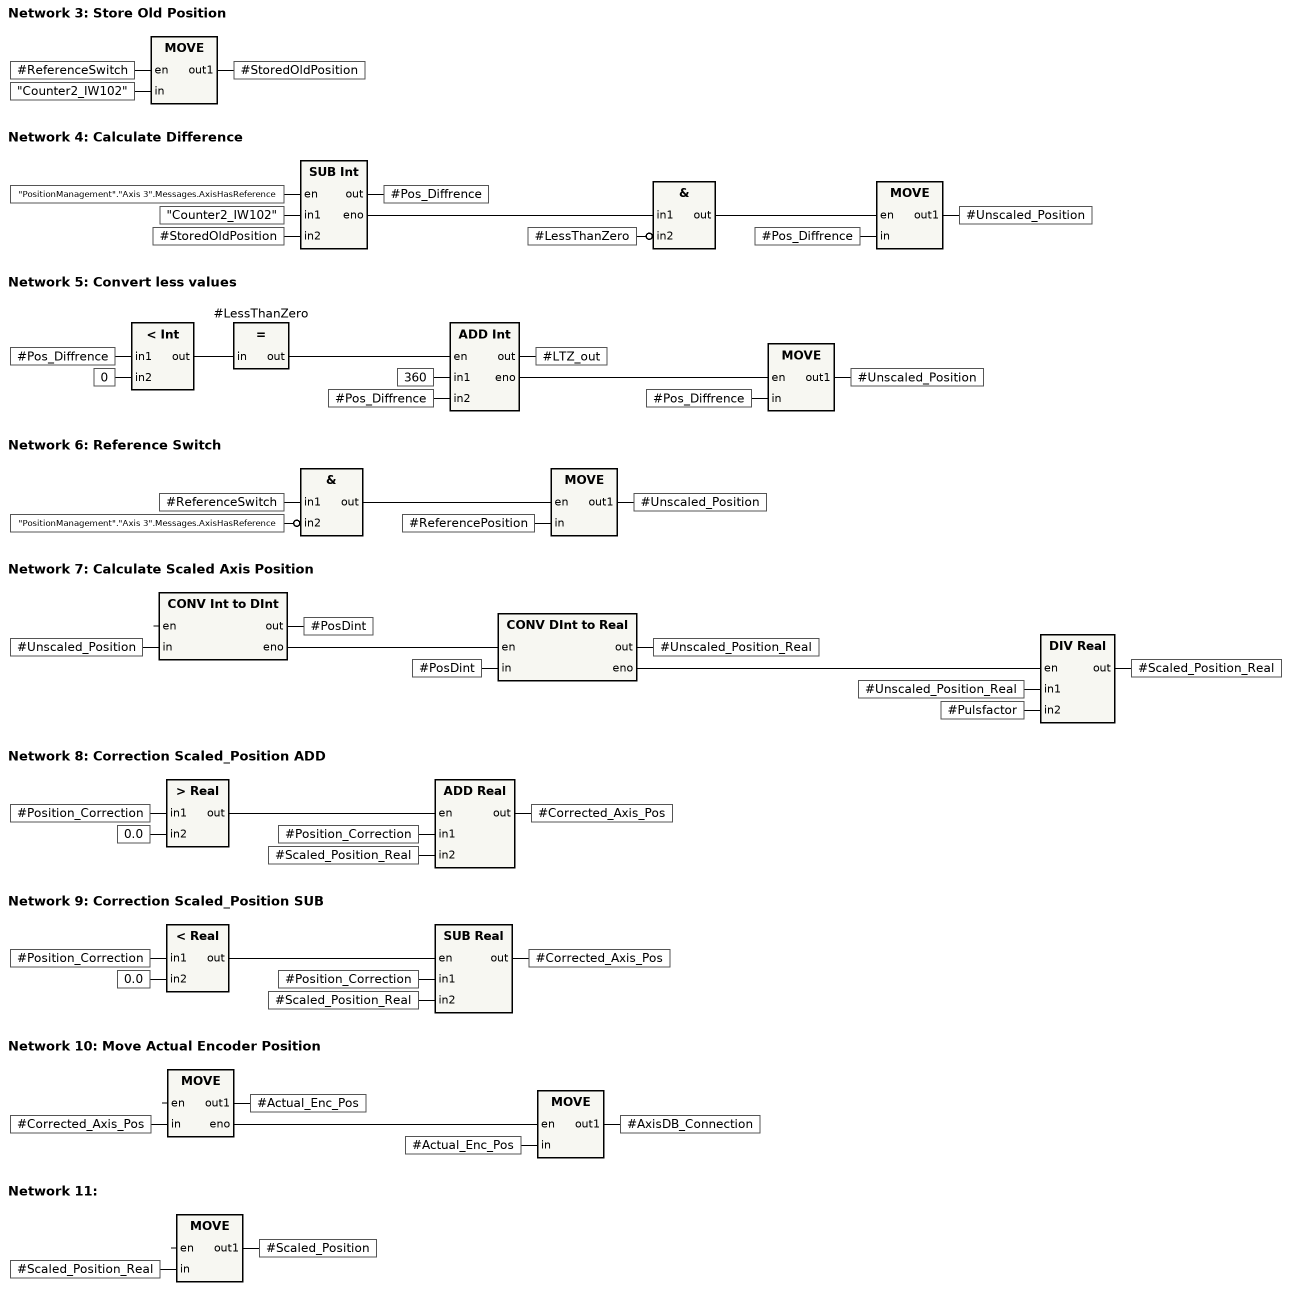
   IF #ReferenceSwitch THEN #StoredOldPosition := "Counter2_IW102"; END_IF;
END_REGION

REGION Network 4: Calculate Difference
   // ENO of a box is taken as its EN; it also drops when the box reports an error
   IF "PositionManagement"."Axis 3".Messages.AxisHasReference THEN
       #Pos_Diffrence := "Counter2_IW102" - #StoredOldPosition;
   END_IF;
   IF "PositionManagement"."Axis 3".Messages.AxisHasReference AND NOT #LessThanZero THEN
       #Unscaled_Position := #Pos_Diffrence;
   END_IF;
END_REGION

REGION Network 5: Convert less values
   // ENO of a box is taken as its EN; it also drops when the box reports an error
   #LessThanZero := #Pos_Diffrence < 0;
   IF #LessThanZero THEN
       #LTZ_out := 360 + #Pos_Diffrence;
       #Unscaled_Position := #Pos_Diffrence;
   END_IF;
END_REGION

REGION Network 6: Reference Switch
   IF #ReferenceSwitch AND NOT "PositionManagement"."Axis 3".Messages.AxisHasReference THEN
       #Unscaled_Position := #ReferencePosition;
   END_IF;
END_REGION

REGION Network 7: Calculate Scaled Axis Position
   // ENO of a box is taken as its EN; it also drops when the box reports an error
   #PosDint := INT_TO_DINT(#Unscaled_Position);
   #Unscaled_Position_Real := DINT_TO_REAL(#PosDint);
   #Scaled_Position_Real := #Unscaled_Position_Real / #Pulsfactor;
END_REGION

REGION Network 8: Correction Scaled_Position ADD
   IF #Position_Correction > 0.0 THEN
       #Corrected_Axis_Pos := #Position_Correction + #Scaled_Position_Real;
   END_IF;
END_REGION

REGION Network 9: Correction Scaled_Position SUB
   IF #Position_Correction < 0.0 THEN
       #Corrected_Axis_Pos := #Position_Correction - #Scaled_Position_Real;
   END_IF;
END_REGION

REGION Network 10: Move Actual Encoder Position
   // ENO of a box is taken as its EN; it also drops when the box reports an error
   #Actual_Enc_Pos := #Corrected_Axis_Pos;
   #AxisDB_Connection := #Actual_Enc_Pos;
END_REGION

REGION Network 11
   #Scaled_Position := #Scaled_Position_Real;
END_REGION
END_FUNCTION

FUNCTION_BLOCK "MC_Move"   // FB10, FBD
TITLE = MC_Move
VERSION : 0.1
// Block moves an Axis to an Desired Position, this block comes with the brake feature. When the axis is on position it keeps the brake for a time. You can set the time in the Brake Time field.
// stored: AutoNumber true, IsIECCheckEnabled false, UDAEnableTagReadback false
   VAR_INPUT
      Start : Bool;
      "Desired Position" : Real;
      "Speed (50-75%)" : Int;
      "Brake on Position" : Bool;
      Acceleration : Real;
      Deacceleration : Real;
      "Drive Ready" : Bool;
      "Drive On Position" : Bool;
      "Brake Time" : Time := T#500ms;
      "Safety OK" : Bool;
   END_VAR
   VAR_OUTPUT
      Go : Bool;
      "Desired Position Out" : Real;
      "Speed Output" : Int;
      "Acceleration Out" : Real;
      "Deacceleration Out" : Real;
      "Brake Out" : Bool;
   END_VAR
   VAR_TEMP
      SR_1 : Bool;
   END_VAR
BEGIN

REGION Network 1: Start - Go To Position + Speed
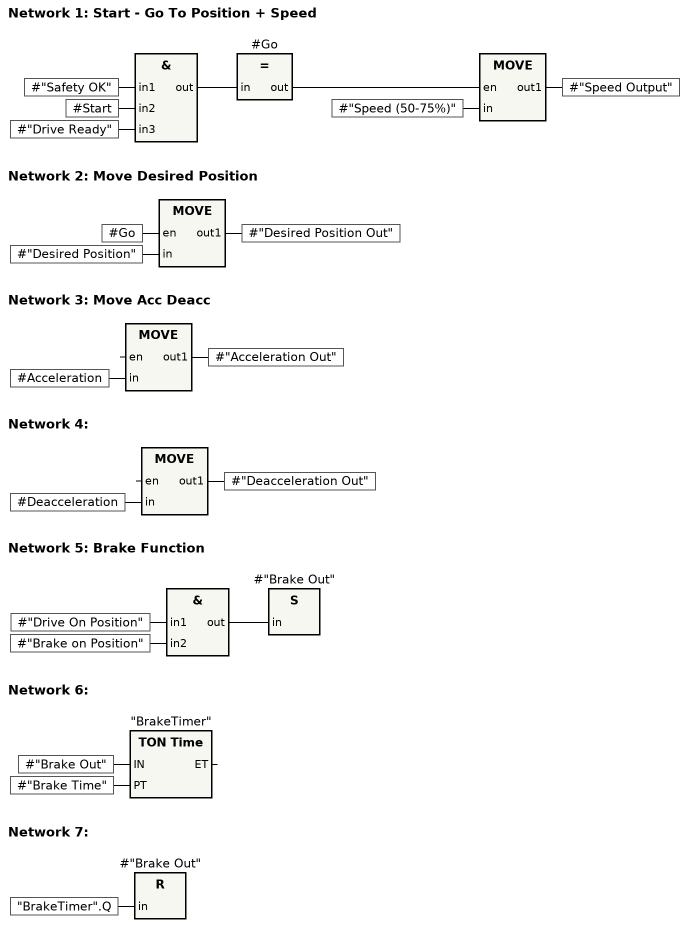
   #Go := #"Safety OK" AND #Start AND #"Drive Ready";
   IF #Go THEN #"Speed Output" := #"Speed (50-75%)"; END_IF;
END_REGION

REGION Network 2: Move Desired Position
   IF #Go THEN #"Desired Position Out" := #"Desired Position"; END_IF;
END_REGION

REGION Network 3: Move Acc Deacc
   #"Acceleration Out" := #Acceleration;
END_REGION

REGION Network 4
   #"Deacceleration Out" := #Deacceleration;
END_REGION

REGION Network 5: Brake Function
   IF #"Drive On Position" AND #"Brake on Position" THEN #"Brake Out" := TRUE; END_IF;
END_REGION

REGION Network 6
   "BrakeTimer".TON(IN := #"Brake Out", PT := #"Brake Time");
END_REGION

REGION Network 7
   IF "BrakeTimer".Q THEN #"Brake Out" := FALSE; END_IF;
END_REGION
END_FUNCTION_BLOCK

FUNCTION_BLOCK "MC_Jog"   // FB11, FBD
TITLE = MC_Jog
VERSION : 0.1
// With this block you can Jog an Axis manual, you can set the speed on 25%, 50% or 75%. It also has an brake functionality, when you set Brake to true, it holds the brake for 2 seconds, then releases it.
// stored: AutoNumber true, IsIECCheckEnabled false, UDAEnableTagReadback false
   VAR_INPUT
      "Jog Forward" : Bool;
      "Jog Backward" : Bool;
      Speed : Int;
      Brake : Bool;
   END_VAR
   VAR_OUTPUT
      "Drive Fwd Output" : Bool;
      "Drive Rev Output" : Bool;
      "Drive Speed Output" : Int;
      "Drive Brake Output" : Bool;
   END_VAR
BEGIN

REGION Network 1: Manual Control
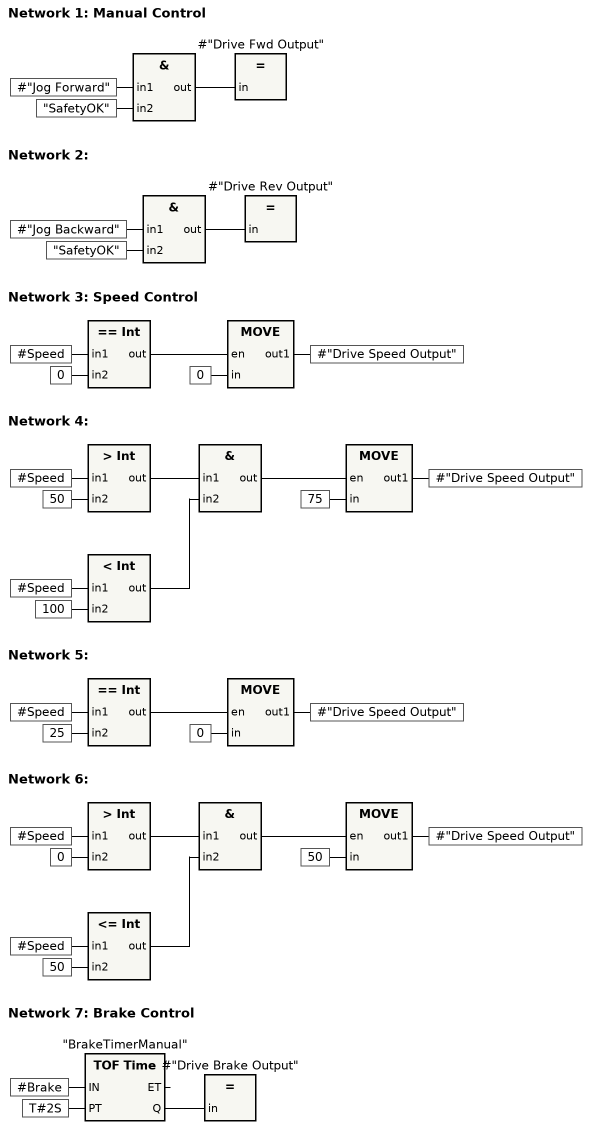
   #"Drive Fwd Output" := #"Jog Forward" AND "SafetyOK";
END_REGION

REGION Network 2
   #"Drive Rev Output" := #"Jog Backward" AND "SafetyOK";
END_REGION

REGION Network 3: Speed Control
   IF #Speed = 0 THEN #"Drive Speed Output" := 0; END_IF;
END_REGION

REGION Network 4
   IF (#Speed > 50) AND (#Speed < 100) THEN #"Drive Speed Output" := 75; END_IF;
END_REGION

REGION Network 5
   IF #Speed = 25 THEN #"Drive Speed Output" := 0; END_IF;
END_REGION

REGION Network 6
   IF (#Speed > 0) AND (#Speed <= 50) THEN #"Drive Speed Output" := 50; END_IF;
END_REGION

REGION Network 7: Brake Control
   "BrakeTimerManual".TOF(IN := #Brake, PT := T#2S);
   #"Drive Brake Output" := "BrakeTimerManual".Q;
END_REGION
END_FUNCTION_BLOCK

FUNCTION_BLOCK "ProductBuffer"
{ S7_Optimized_Access := 'FALSE' }
VERSION : 0.1
   VAR_INPUT 
      SensorInput : Bool;
      TimeDelay : Time;
      TriggerFeedback : Bool;
   END_VAR

   VAR_OUTPUT 
      TriggerMovement : Bool;
      ProductCount : Int;
   END_VAR

   VAR 
      PrevSensor : Bool;
      DelayTimer {InstructionName := 'TON'; LibVersion := '1.0'; S7_SetPoint := 'False'} : TON;
      MovementActive { S7_SetPoint := 'True'} : Bool;
   END_VAR


BEGIN
	// Flankdetectie op sensor
	IF #SensorInput AND NOT #PrevSensor THEN
	    IF #ProductCount < 32767 THEN
	        #ProductCount := #ProductCount + 1;
	    END_IF;
	END_IF;
	#PrevSensor := #SensorInput;
	
	// Timer mag alleen lopen als:
	// - Er producten zijn
	// - Er geen beweging actief is
	IF (#ProductCount > 0) AND (NOT #MovementActive) THEN
	    #DelayTimer(IN := TRUE,
	                PT := #TimeDelay);
	ELSE
	    #DelayTimer(IN := FALSE,
	                PT := #TimeDelay);
	END_IF;
	
	// Als de timer klaar is → activeer beweging en zet MovementActive
	IF #DelayTimer.Q THEN
	    #TriggerMovement := TRUE;
	    #MovementActive := TRUE;
	    #ProductCount := #ProductCount - 1;
	    #DelayTimer(IN := FALSE,
	                PT := #TimeDelay); // Reset timer
	END_IF;
	
	// Wacht op TriggerFeedback om TriggerMovement terug laag te zetten
	IF #MovementActive AND #TriggerFeedback THEN
	    #TriggerMovement := FALSE;
	    #MovementActive := FALSE;
	END_IF;
	
END_FUNCTION_BLOCK

FUNCTION_BLOCK "ProductBuffer_V3"
{ S7_Optimized_Access := 'FALSE' }
VERSION : 0.1
   VAR_INPUT 
      SensorInput : Bool;   // Sensor aan begin band
      EncoderPosition : DInt;   // Koppel aan Encoder Data Instance
      TriggerDistance : DInt;   // Gewenste Afstand Product voor trigger
      TriggerFeedback : Bool;
   END_VAR

   VAR_OUTPUT 
      TriggerMovement : Bool;   // Trigger Start Movement
      ProductCount : Int;   // Count products in buffer
   END_VAR

   VAR 
      ProductBuffer { S7_SetPoint := 'False'} : Array[0..9] of "ProductTrack";
      PrevSensor { S7_SetPoint := 'True'} : Bool;
      MovementActive : Bool;
      i : Int;
      Distance : DInt;
   END_VAR


BEGIN
	// 1️⃣ Flankdetectie - detecteer nieuw product
	IF #SensorInput AND NOT #PrevSensor THEN
	    FOR #i := 0 TO 9 DO
	        IF NOT #ProductBuffer[#i].Active THEN
	            #ProductBuffer[#i].StartPosition := #EncoderPosition;
	            #ProductBuffer[#i].Active := TRUE;
	            EXIT;
	        END_IF;
	    END_FOR;
	END_IF;
	#PrevSensor := #SensorInput;
	
	// 2️⃣ Tel actieve producten
	#ProductCount := 0;
	FOR #i := 0 TO 9 DO
	    IF #ProductBuffer[#i].Active THEN
	        #ProductCount := #ProductCount + 1;
	    END_IF;
	END_FOR;
	
	// 3️⃣ Zoek eerste product dat zijn afstand heeft afgelegd
	IF NOT #MovementActive THEN
	    FOR #i := 0 TO 9 DO
	        IF #ProductBuffer[#i].Active THEN
	            #Distance := #ProductBuffer[#i].StartPosition - #EncoderPosition;
	            IF #Distance >= #TriggerDistance THEN
	                #TriggerMovement := TRUE;
	                #MovementActive := TRUE;
	                #ProductBuffer[#i].Active := FALSE;
	                EXIT;
	            END_IF;
	        END_IF;
	    END_FOR;
	END_IF;
	
	// 4️⃣ Wacht op feedback om beweging af te ronden
	IF #MovementActive AND #TriggerFeedback THEN
	    #TriggerMovement := FALSE;
	    #MovementActive := FALSE;
	END_IF;
	
END_FUNCTION_BLOCK

FUNCTION_BLOCK "FB_EncoderFeedback_Lineair"   // FB21, FBD
TITLE = Encoder Feedback Function Block Lineair Axis
VERSION : 0.1
// stored: AutoNumber true, IsIECCheckEnabled false, UDAEnableTagReadback false
   VAR_INPUT
      CounterTag { ExternalVisible := 'False'; ExternalWritable := 'False'} : DInt;   // Connect to the CounterTag IW102
      Position_Offset { ExternalVisible := 'False'; ExternalWritable := 'False'} : Real;   // Fill in the tolerance, when the axis approves the position. Above or below the desired position
      Pulsfactor { ExternalVisible := 'False'; ExternalWritable := 'False'} : Real;   // Number of pulses after an defined distance of the axis.
      Position_Correction { ExternalVisible := 'False'; ExternalWritable := 'False'} : Real;   // Small Position Correction for the Axis
      ReferenceRun_Command { ExternalVisible := 'False'; ExternalWritable := 'False'} : Bool;   // Command of starting the referencerun
      ReferenceSwitch { ExternalVisible := 'False'; ExternalWritable := 'False'} : Bool;   // ReferenceSwitch Mounted on Axis
      ReferencePosition { ExternalVisible := 'False'; ExternalWritable := 'False'} : Int;   // Position where the index puls of the reference switch enters.
      WrappingPosition : Real;   // Max Position of the axis. From there the position
   END_VAR
   VAR_OUTPUT
      Scaled_Position { ExternalVisible := 'False'; ExternalWritable := 'False'} : Real;   // Scaled Position scaled with Pulsfactor
      Actual_Enc_Pos { ExternalVisible := 'False'; ExternalWritable := 'False'} : Real;   // Actual Encoder Position
      AxisDB_Connection { ExternalVisible := 'False'; ExternalWritable := 'False'} : Real;   // Connection with Axis DB connection
   END_VAR
   VAR_TEMP
      Corrected_Axis_Pos : Real;
      Unscaled_Position : DInt;   // Unscaled Position of the Encoder
      Unsc2 : DInt;   // Unsc 2 position
      Act_Enc_Pos_Int : DInt;
      Scaled_Position_Real : Real;
      PosDint : DInt;
      Unscaled_Position_Real : Real;
      InternalCounter : DInt;
      CalDifCounter : DInt;
      Pos_Storage : DInt;
      Pos_Diffrence : DInt;
      Add_Pos : DInt;
      Sub_Pos : DInt;
      LessThanZero : Bool;
      LTZ_out : DInt;
      WrappedPosTemp : Real;
      DivWrapping : Real;
      TruncWrapping : DInt;
      TruncWrappingReal : Real;
      ScaledBackWrapping : Real;
      AxisPosTooHigh : Bool;
      WeDontUseThisAnymore : Bool;
      SRMOve : Bool;
      noreset : Bool;
      nououtput : Bool;
      OverflowProtectPulses : DInt;
      SegmentCounter : DInt;
   END_VAR
BEGIN

REGION Network 1: Overflow Buffer FB
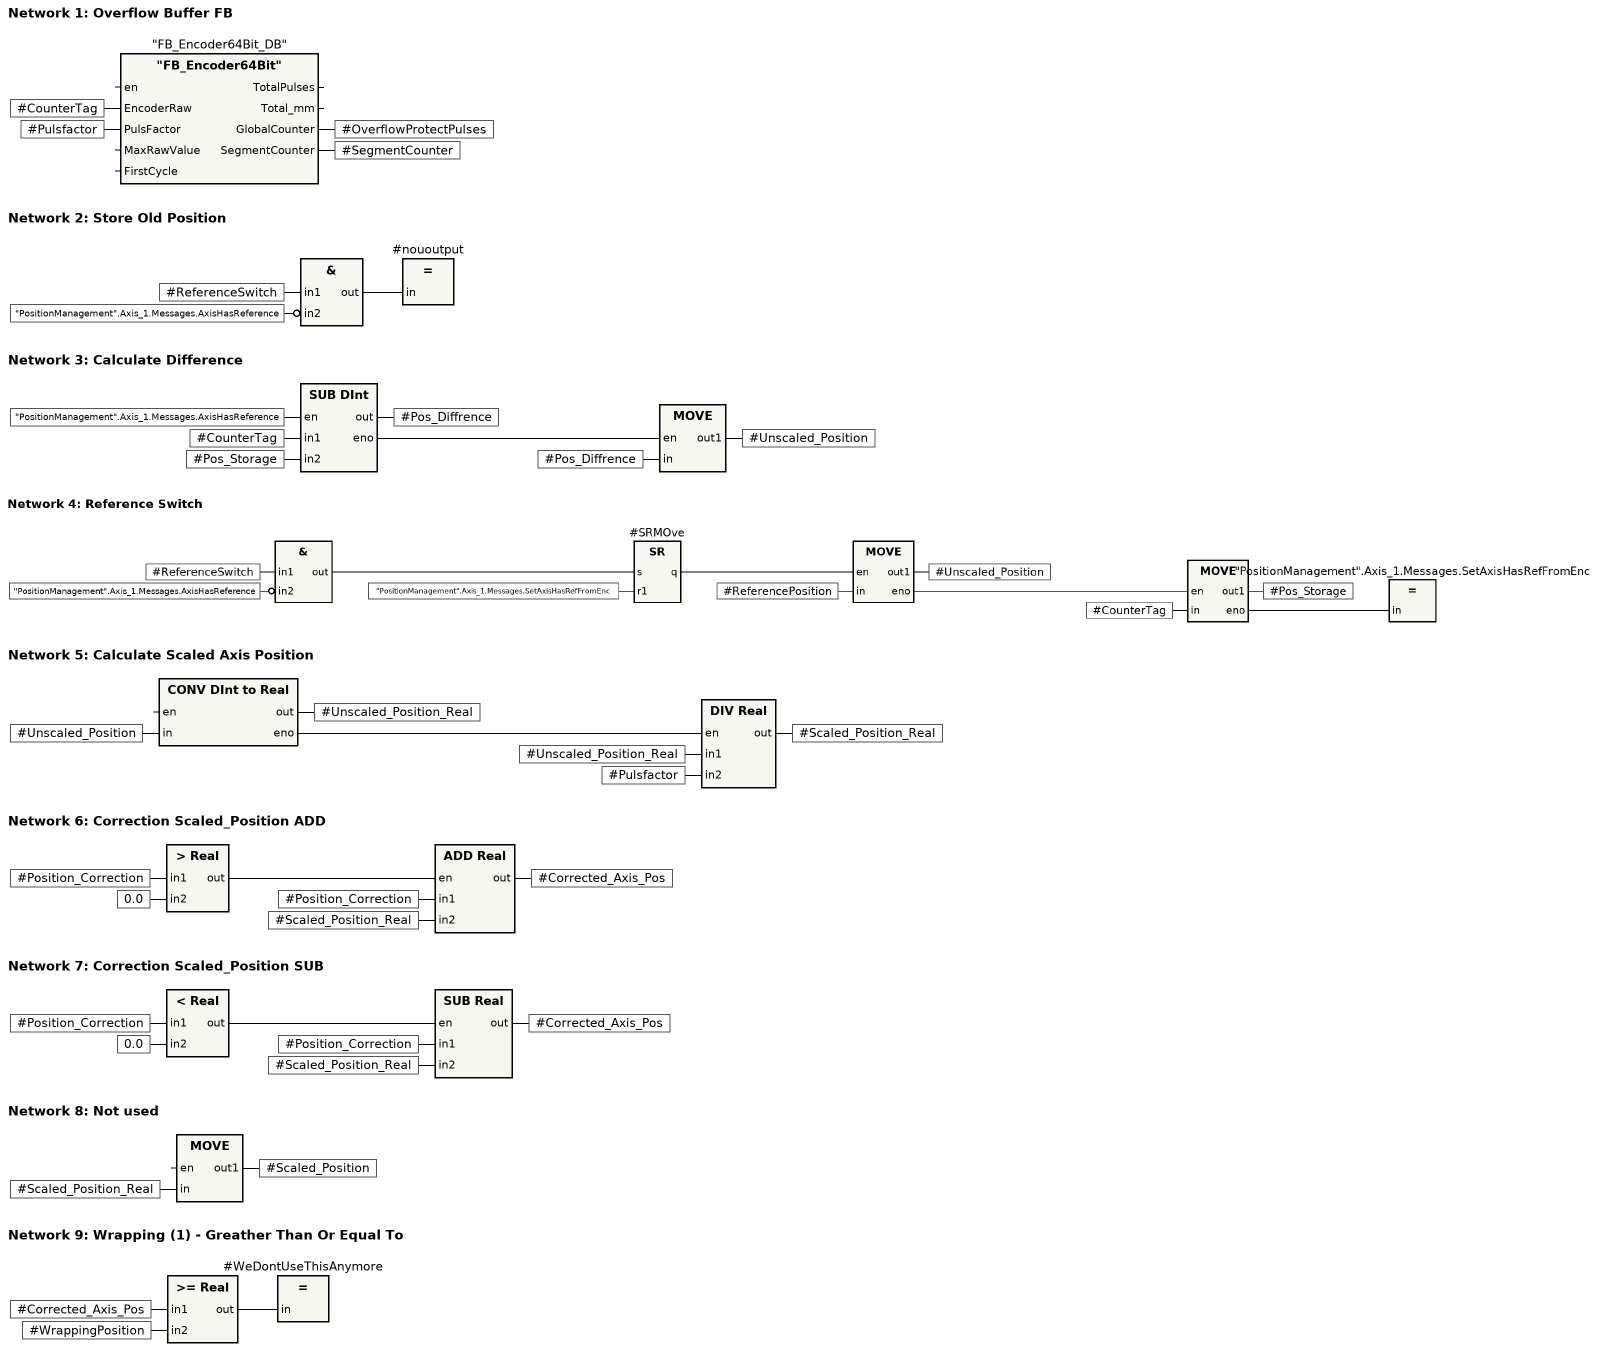
   "FB_Encoder64Bit_DB"(EncoderRaw := #CounterTag,   // "FB_Encoder64Bit"
                        PulsFactor := #Pulsfactor,
                        GlobalCounter => #OverflowProtectPulses,
                        SegmentCounter => #SegmentCounter);
END_REGION

REGION Network 2: Store Old Position
   #nououtput := #ReferenceSwitch AND NOT "PositionManagement".Axis_1.Messages.AxisHasReference;
END_REGION

REGION Network 3: Calculate Difference
   // ENO of a box is taken as its EN; it also drops when the box reports an error
   IF "PositionManagement".Axis_1.Messages.AxisHasReference THEN
       #Pos_Diffrence := #CounterTag - #Pos_Storage;
       #Unscaled_Position := #Pos_Diffrence;
   END_IF;
END_REGION

REGION Network 4: Reference Switch
   // ENO of a box is taken as its EN; it also drops when the box reports an error
   IF #ReferenceSwitch AND NOT "PositionManagement".Axis_1.Messages.AxisHasReference THEN
       #SRMOve := TRUE;   // SR flip-flop
   END_IF;
   IF "PositionManagement".Axis_1.Messages.SetAxisHasRefFromEnc THEN #SRMOve := FALSE; END_IF;
   IF #SRMOve THEN
       #Unscaled_Position := #ReferencePosition;
       #Pos_Storage := #CounterTag;
   END_IF;
   "PositionManagement".Axis_1.Messages.SetAxisHasRefFromEnc := #SRMOve;
END_REGION

REGION Network 5: Calculate Scaled Axis Position
   // ENO of a box is taken as its EN; it also drops when the box reports an error
   #Unscaled_Position_Real := DINT_TO_REAL(#Unscaled_Position);
   #Scaled_Position_Real := #Unscaled_Position_Real / #Pulsfactor;
END_REGION

REGION Network 6: Correction Scaled_Position ADD
   IF #Position_Correction > 0.0 THEN
       #Corrected_Axis_Pos := #Position_Correction + #Scaled_Position_Real;
   END_IF;
END_REGION

REGION Network 7: Correction Scaled_Position SUB
   IF #Position_Correction < 0.0 THEN
       #Corrected_Axis_Pos := #Position_Correction - #Scaled_Position_Real;
   END_IF;
END_REGION

REGION Network 8: Not used
   #Scaled_Position := #Scaled_Position_Real;
END_REGION

REGION Network 9: Wrapping (1) - Greather Than Or Equal To
   #WeDontUseThisAnymore := #Corrected_Axis_Pos >= #WrappingPosition;
END_REGION

REGION Network 10: Wrapping (2) - MOVE Axis Pos Too High
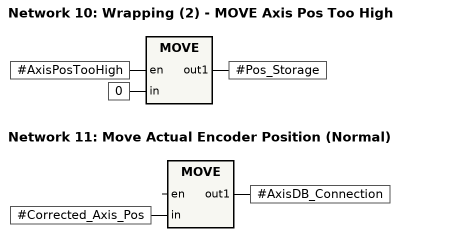
   IF #AxisPosTooHigh THEN #Pos_Storage := 0; END_IF;
END_REGION

REGION Network 11: Move Actual Encoder Position (Normal)
   #AxisDB_Connection := #Corrected_Axis_Pos;
END_REGION
END_FUNCTION_BLOCK

FUNCTION_BLOCK "FB_Encoder64Bit"
{ S7_Optimized_Access := 'FALSE' }
VERSION : 0.1
   VAR_INPUT 
      EncoderRaw : DInt;   // // Ruwe encoderwaarde van hardware (%ID112)
      PulsFactor : Real;
      MaxRawValue : DInt := 20000;
      FirstCycle { ExternalVisible := 'False'; ExternalWritable := 'False'} : Bool := true;
   END_VAR

   VAR_OUTPUT 
      TotalPulses : DInt;
      Total_mm : Real;
      GlobalCounter : DInt;
      SegmentCounter : DInt;
   END_VAR

   VAR_TEMP 
      Delta : DInt;
      LastEncoder_2 : DInt;
      InternalSum_2 : DInt;
      LastEncoder : DInt;
      InternalSum : DInt;
      InternalCount : DInt;
      Delta64 : Int;
      Global_mm : Real;
      Segment_mm : Real;
   END_VAR

   VAR CONSTANT 
      OverflowLimit : DInt := 2000000000;   // // Ondergrens van veilige DINT-waarde
   END_VAR


BEGIN
	// Init
	IF #FirstCycle THEN
	    #LastEncoder := #EncoderRaw;
	    #FirstCycle := FALSE;
	END_IF;
	
	// Delta berekenen
	#Delta := #EncoderRaw - #LastEncoder;
	
	// Gebruik waarden binnen DINT-bereik
	// Corrigeer overflow (positief → negatief)
	IF #Delta > 1000000000 THEN
	    #Delta := #Delta - 2147483647;
	    #Delta := #Delta - 2147483647; // 2x max DINT
	    #Delta := #Delta - 2; // totaal 4294967296
	END_IF;
	
	// Corrigeer onderflow (negatief → positief)
	IF #Delta < -1000000000 THEN
	    #Delta := #Delta + 2147483647;
	    #Delta := #Delta + 2147483647;
	    #Delta := #Delta + 2;
	END_IF;
	
	// Teller bijwerken
	#InternalCount := #InternalCount + #Delta;
	#LastEncoder := #EncoderRaw;
	
	// Output absolute teller
	#GlobalCounter := #InternalCount;
	#Global_mm := DINT_TO_REAL(#GlobalCounter) * #PulsFactor;
	
	// Segmentpositie berekenen (positief binnen 0..MaxRawValue)
	#SegmentCounter := #InternalCount MOD #MaxRawValue;
	IF #SegmentCounter < 0 THEN
	    #SegmentCounter := #SegmentCounter + #MaxRawValue;
	END_IF;
	
	#Segment_mm := DINT_TO_REAL(#SegmentCounter) * #PulsFactor;
END_FUNCTION_BLOCK

FUNCTION "8 - Noodsleutel" : Void   // FC9, LAD
TITLE = Emergency Switch
VERSION : 0.1
// stored: AutoNumber true, IsIECCheckEnabled false, UDAEnableTagReadback false
BEGIN

REGION Network 1
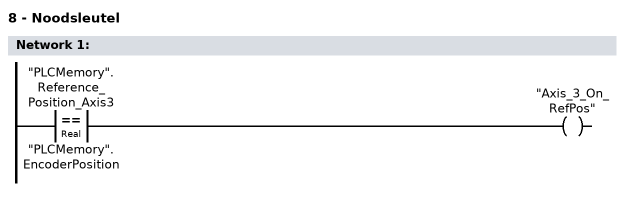
   RUNG wire#powerrail
      { S7_Templates := "SrcType := Real" } EQ_Contact(in1 := "PLCMemory".Reference_Position_Axis3, in2 := "PLCMemory".EncoderPosition)
      Coil( "Axis_3_On_RefPos" )
   END_RUNG
   // the same network as SCL:
   "Axis_3_On_RefPos" := "PLCMemory".Reference_Position_Axis3 = "PLCMemory".EncoderPosition;
END_REGION
END_FUNCTION

FUNCTION_BLOCK "Programma 1 - Test"   // FB12, GRAPH
VERSION : 0.1
// stored: AcknowledgeErrorsRequired true, AutoNumber true, CreateMinimizedDB false, IsIECCheckEnabled false, LanguageInNetworks LAD, LockOperatingMode false, PermanentILProcessingInMANMode false, SkipSteps false, UDAEnableTagReadback false, WithAlarmHandling true
   VAR_INPUT
      OFF_SQ { ExternalAccessible := 'False'; ExternalVisible := 'False'; ExternalWritable := 'False'} : Bool := false;   // Turn sequence off
      INIT_SQ { ExternalAccessible := 'False'; ExternalVisible := 'False'; ExternalWritable := 'False'} : Bool := false;   // Set sequence to initial state
      ACK_EF { ExternalAccessible := 'False'; ExternalVisible := 'False'; ExternalWritable := 'False'} : Bool := false;   // Acknowledge all errors and faults
      S_PREV { ExternalAccessible := 'False'; ExternalVisible := 'False'; ExternalWritable := 'False'} : Bool := false;   // Output previous step in parameter S_NO
      S_NEXT { ExternalAccessible := 'False'; ExternalVisible := 'False'; ExternalWritable := 'False'} : Bool := false;   // Indicate next step in parameter S_NO
      SW_AUTO { ExternalAccessible := 'False'; ExternalVisible := 'False'; ExternalWritable := 'False'} : Bool := false;   // Automatic mode
      SW_TAP { ExternalAccessible := 'False'; ExternalVisible := 'False'; ExternalWritable := 'False'} : Bool := false;   // Semiautomatic/switch with transition
      SW_TOP { ExternalAccessible := 'False'; ExternalVisible := 'False'; ExternalWritable := 'False'} : Bool := false;   // Semiautomatic/ignore transition
      SW_MAN { ExternalAccessible := 'False'; ExternalVisible := 'False'; ExternalWritable := 'False'} : Bool := false;   // Manual mode
      S_SEL { ExternalAccessible := 'False'; ExternalVisible := 'False'; ExternalWritable := 'False'} : Int := 0;   // Select step to be output to S_NO
      S_ON { ExternalAccessible := 'False'; ExternalVisible := 'False'; ExternalWritable := 'False'} : Bool := false;   // Activate step indicated in S_NO
      S_OFF { ExternalAccessible := 'False'; ExternalVisible := 'False'; ExternalWritable := 'False'} : Bool := false;   // Deactivate step indicated S_NO
      T_PUSH { ExternalAccessible := 'False'; ExternalVisible := 'False'; ExternalWritable := 'False'} : Bool := false;   // Enable transition to switch in semi automatic mode
      "Confimation Position 1" : Bool;
      "Confirmation Position 2" : Bool;
      "Products more than zero" : Bool;
      "Products zero" : Bool;
      "Timer 1" : Time;
   END_VAR
   VAR_OUTPUT
      S_NO { ExternalAccessible := 'False'; ExternalVisible := 'False'; ExternalWritable := 'False'} : Int := 0;   // Step number
      S_MORE { ExternalAccessible := 'False'; ExternalVisible := 'False'; ExternalWritable := 'False'} : Bool := false;   // More steps are available and can be shown in S_NO
      S_ACTIVE { ExternalAccessible := 'False'; ExternalVisible := 'False'; ExternalWritable := 'False'} : Bool := false;   // Step indicated in S_NO is active
      ERR_FLT { ExternalAccessible := 'False'; ExternalVisible := 'False'; ExternalWritable := 'False'} : Bool := false;   // Interlock or supervision group error
      AUTO_ON { ExternalAccessible := 'False'; ExternalVisible := 'False'; ExternalWritable := 'False'} : Bool := false;   // Automatic mode is active
      TAP_ON { ExternalAccessible := 'False'; ExternalVisible := 'False'; ExternalWritable := 'False'} : Bool := false;   // Semiautomatic mode/step with transition enabled
      TOP_ON { ExternalAccessible := 'False'; ExternalVisible := 'False'; ExternalWritable := 'False'} : Bool := false;   // Semiautomatic mode/ignore transition enabled
      MAN_ON { ExternalAccessible := 'False'; ExternalVisible := 'False'; ExternalWritable := 'False'} : Bool := false;   // Manual mode is active
      "Move Position 1" : Bool;
      "Move Position 2" : Bool;
   END_VAR
   VAR DB_SPECIFIC
      S_DISPLAY { ExternalAccessible := 'False'; ExternalVisible := 'False'; ExternalWritable := 'False'} : Int;   // Internal display of output parameter S_NO
      S_SEL_OLD { ExternalAccessible := 'False'; ExternalVisible := 'False'; ExternalWritable := 'False'} : Int;   // Previous value in S_SEL
      S_DISPIDX { ExternalAccessible := 'False'; ExternalVisible := 'False'; ExternalWritable := 'False'} : Byte;   // Index of the step in S_NO
      T_DISPIDX { ExternalAccessible := 'False'; ExternalVisible := 'False'; ExternalWritable := 'False'} : Byte;   // Index of the transition displayed in T_NO
      MOP { ExternalAccessible := 'False'; ExternalVisible := 'False'; ExternalWritable := 'False'} : Struct   // Mode
         AUTO { ExternalAccessible := 'False'; ExternalVisible := 'False'; ExternalWritable := 'False'} : Bool := true;   // Status: automatic mode
         MAN { ExternalAccessible := 'False'; ExternalVisible := 'False'; ExternalWritable := 'False'} : Bool := false;   // Status: manual mode
         TAP { ExternalAccessible := 'False'; ExternalVisible := 'False'; ExternalWritable := 'False'} : Bool := false;   // Status: semi automatic/switch with transition
         TOP { ExternalAccessible := 'False'; ExternalVisible := 'False'; ExternalWritable := 'False'} : Bool := false;   // Status: semi automatic/ignore transition
         ACK_S { ExternalAccessible := 'False'; ExternalVisible := 'False'; ExternalWritable := 'False'} : Bool := false;   // Request: acknowledge step at parameter S_NO
         REG_S { ExternalAccessible := 'False'; ExternalVisible := 'False'; ExternalWritable := 'False'} : Bool := false;   // Request: register step indicated in S_NO
         T_PREV { ExternalAccessible := 'False'; ExternalVisible := 'False'; ExternalWritable := 'False'} : Bool := false;   // Request: output previous valid transition in T_NO
         T_NEXT { ExternalAccessible := 'False'; ExternalVisible := 'False'; ExternalWritable := 'False'} : Bool := false;   // Request: output next valid transition in T_NO
         LOCK { ExternalAccessible := 'False'; ExternalVisible := 'False'; ExternalWritable := 'False'} : Bool := true;   // Status: interlocks activated
         SUP { ExternalAccessible := 'False'; ExternalVisible := 'False'; ExternalWritable := 'False'} : Bool := true;   // Status: supervisions activated
         ACKREQ { ExternalAccessible := 'False'; ExternalVisible := 'False'; ExternalWritable := 'False'} : Bool := true;   // Status: acknowledgment required
         SSKIP { ExternalAccessible := 'False'; ExternalVisible := 'False'; ExternalWritable := 'False'} : Bool := false;   // Status: "Skip steps" enabled
         OFF { ExternalAccessible := 'False'; ExternalVisible := 'False'; ExternalWritable := 'False'} : Bool := false;   // Request: deactivate all steps
         INIT { ExternalAccessible := 'False'; ExternalVisible := 'False'; ExternalWritable := 'False'} : Bool := true;   // Request: set sequence to initial state
         HALT { ExternalAccessible := 'False'; ExternalVisible := 'False'; ExternalWritable := 'False'} : Bool := false;   // Status: sequence halted
         TMS_HALT { ExternalAccessible := 'False'; ExternalVisible := 'False'; ExternalWritable := 'False'} : Bool := false;   // Status: all internal timers held
         OPS_ZERO { ExternalAccessible := 'False'; ExternalVisible := 'False'; ExternalWritable := 'False'} : Bool := false;   // Status: set all operands processed with N, L, D instructions to 0
         SACT_DISP { ExternalAccessible := 'False'; ExternalVisible := 'False'; ExternalWritable := 'False'} : Bool := true;   // Status: display active steps only
         SEF_DISP { ExternalAccessible := 'False'; ExternalVisible := 'False'; ExternalWritable := 'False'} : Bool := false;   // Status: display only steps with errors and disrupted steps
         SALL_DISP { ExternalAccessible := 'False'; ExternalVisible := 'False'; ExternalWritable := 'False'} : Bool := false;   // Status: display all steps
         S_PREV { ExternalAccessible := 'False'; ExternalVisible := 'False'; ExternalWritable := 'False'} : Bool := false;   // Request: output previous step to S_NO
         S_NEXT { ExternalAccessible := 'False'; ExternalVisible := 'False'; ExternalWritable := 'False'} : Bool := false;   // Request: Output next step at S_NO parameter
         S_SELOK { ExternalAccessible := 'False'; ExternalVisible := 'False'; ExternalWritable := 'False'} : Bool := false;   // Request: output step number from S_SEL to S_NO
         S_ON { ExternalAccessible := 'False'; ExternalVisible := 'False'; ExternalWritable := 'False'} : Bool := false;   // Request: activate step indicated in S_NO
         S_OFF { ExternalAccessible := 'False'; ExternalVisible := 'False'; ExternalWritable := 'False'} : Bool := false;   // Request: deactivate step at parameter S_NO
         T_PUSH { ExternalAccessible := 'False'; ExternalVisible := 'False'; ExternalWritable := 'False'} : Bool := false;   // Request: transition switching enabled
         REG { ExternalAccessible := 'False'; ExternalVisible := 'False'; ExternalWritable := 'False'} : Bool := false;   // Request: register all interlock and supervision errors
         ACK { ExternalAccessible := 'False'; ExternalVisible := 'False'; ExternalWritable := 'False'} : Bool := false;   // Request: acknowledge all interlock and supervision errors
         IL_PERM { ExternalAccessible := 'False'; ExternalVisible := 'False'; ExternalWritable := 'False'} : Bool := false;   // Status: permanent processing of all interlocks
         T_PERM { ExternalAccessible := 'False'; ExternalVisible := 'False'; ExternalWritable := 'False'} : Bool := false;   // Status: permanent processing of all transitions
         ILP_MAN { ExternalAccessible := 'False'; ExternalVisible := 'False'; ExternalWritable := 'False'} : Bool := false;   // Status: permanent processing of all interlocks in manual mode
      END_STRUCT;
      TICKS { ExternalAccessible := 'False'; ExternalVisible := 'False'; ExternalWritable := 'False'} : Struct   // Clock speeds
         DELTA { ExternalAccessible := 'False'; ExternalVisible := 'False'; ExternalWritable := 'False'} : Time := T#0ms;   // Time difference between cycles
         OLD { ExternalAccessible := 'False'; ExternalVisible := 'False'; ExternalWritable := 'False'} : Time := T#0ms;   // 10 ms clock counter value in last cycle
         NEW { ExternalAccessible := 'False'; ExternalVisible := 'False'; ExternalWritable := 'False'} : Time := T#0ms;   // 10 ms clock counter value in this cycle
      END_STRUCT;
      SQ_FLAGS { ExternalAccessible := 'False'; ExternalVisible := 'False'; ExternalWritable := 'False'} : Struct   // Sequence bit memory
         ERR_FLT { ExternalAccessible := 'False'; ExternalVisible := 'False'; ExternalWritable := 'False'} : Bool := false;   // Interlock and supervision group error
         ERROR { ExternalAccessible := 'False'; ExternalVisible := 'False'; ExternalWritable := 'False'} : Bool := false;   // Interlock group error
         FAULT { ExternalAccessible := 'False'; ExternalVisible := 'False'; ExternalWritable := 'False'} : Bool := false;   // Supervision group error
         RT_FAIL { ExternalAccessible := 'False'; ExternalVisible := 'False'; ExternalWritable := 'False'} : Bool := false;   // Runtime error
         NO_SNO { ExternalAccessible := 'False'; ExternalVisible := 'False'; ExternalWritable := 'False'} : Bool := false;   // Requested step number not found
         NF_OFL { ExternalAccessible := 'False'; ExternalVisible := 'False'; ExternalWritable := 'False'} : Bool := false;   // Overflow: too many ON or OFF requests
         SA_OFL { ExternalAccessible := 'False'; ExternalVisible := 'False'; ExternalWritable := 'False'} : Bool := false;   // Overflow: too many steps active
         TV_OFL { ExternalAccessible := 'False'; ExternalVisible := 'False'; ExternalWritable := 'False'} : Bool := false;   // Overflow: too many valid transitions
         MSG_OFL { ExternalAccessible := 'False'; ExternalVisible := 'False'; ExternalWritable := 'False'} : Bool := false;   // Overflow: not enough system resources for ALARM_S
         NO_SWI { ExternalAccessible := 'False'; ExternalVisible := 'False'; ExternalWritable := 'False'} : Bool := false;   // Do not switch in this cycle
         CYC_OP { ExternalAccessible := 'False'; ExternalVisible := 'False'; ExternalWritable := 'False'} : Bool := false;   // Cyclic execution of the sequence after initialization
         AS_MSG { ExternalAccessible := 'False'; ExternalVisible := 'False'; ExternalWritable := 'False'} : Bool := true;   // Alarms during runtime enabled or disabled by instruction
         AS_SEND { ExternalAccessible := 'False'; ExternalVisible := 'False'; ExternalWritable := 'False'} : Bool := false;   // Send alarms from WR_USMSG or only enter in diagnostics buffer
         SQ_BUSY { ExternalAccessible := 'False'; ExternalVisible := 'False'; ExternalWritable := 'False'} : Bool := false;   // Internal edge memory bit for sequence processing
         SA_BUSY { ExternalAccessible := 'False'; ExternalVisible := 'False'; ExternalWritable := 'False'} : Bool := false;   // Internal edge memory bit for sequence processing
         AS_SIG { ExternalAccessible := 'False'; ExternalVisible := 'False'; ExternalWritable := 'False'} : Bool := false;   // Edge memory bit for alarms from Alarm_S and Alarm_SQ
      END_STRUCT;
   END_VAR
BEGIN
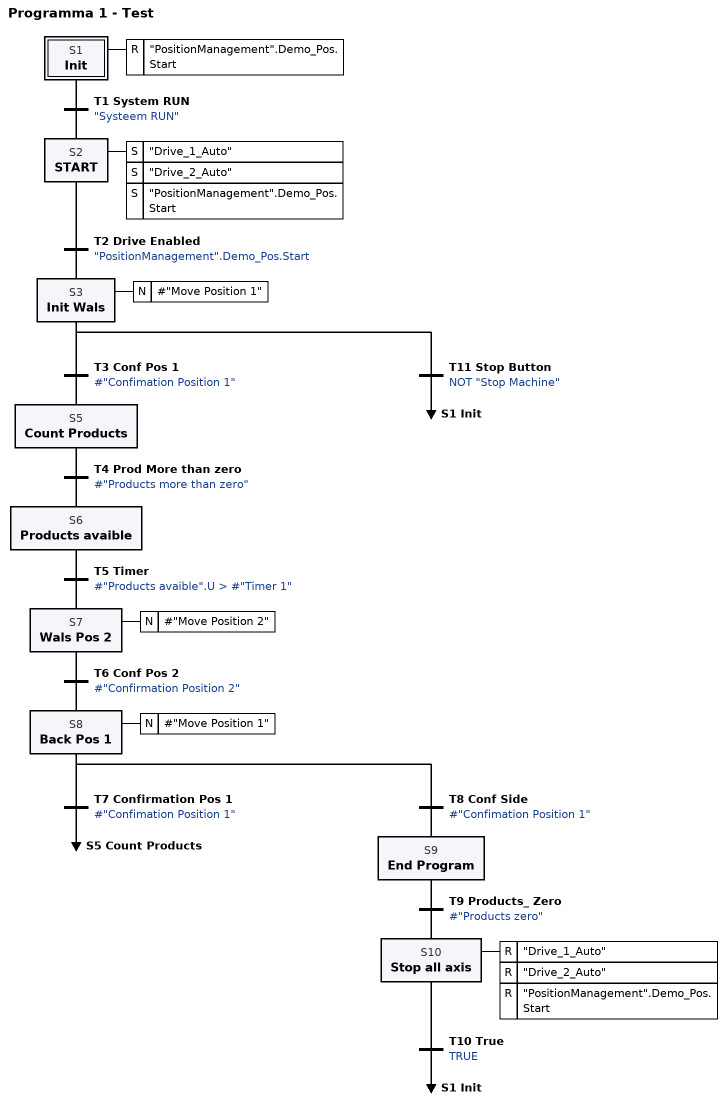
   // sequencer 1: SFC Program
   INITIAL_STEP Init:   // S1
              R    "PositionManagement".Demo_Pos.Start
   END_STEP
   TRANSITION "System RUN" FROM Init TO START   // T1
      := "Systeem RUN";
   END_TRANSITION
   STEP START:   // S2
      // Set Ouputs
              S    "Drive_1_Auto"
              S    "Drive_2_Auto"
              S    "PositionManagement".Demo_Pos.Start
   END_STEP
   TRANSITION "Drive Enabled" FROM START TO "Init Wals"   // T2
      := "PositionManagement".Demo_Pos.Start;
   END_TRANSITION
   STEP "Init Wals":   // S3
      // Move Start Position4
              N    #"Move Position 1"
   END_STEP
   TRANSITION "Conf Pos 1" FROM "Init Wals" TO "Count Products"   // T3
      := #"Confimation Position 1";
   END_TRANSITION
   TRANSITION "Stop Button" FROM "Init Wals" TO Init   // T11, jump
      := NOT "Stop Machine";
   END_TRANSITION
   STEP "Count Products":   // S5
   END_STEP
   TRANSITION "Prod More than zero" FROM "Count Products" TO "Products avaible"   // T4
      := #"Products more than zero";
   END_TRANSITION
   STEP "Products avaible":   // S6
   END_STEP
   TRANSITION "Timer" FROM "Products avaible" TO "Wals Pos 2"   // T5: Timer 1
      := #"Products avaible".U > #"Timer 1";
   END_TRANSITION
   STEP "Wals Pos 2":   // S7
              N    #"Move Position 2"
   END_STEP
   TRANSITION "Conf Pos 2" FROM "Wals Pos 2" TO "Back Pos 1"   // T6
      := #"Confirmation Position 2";
   END_TRANSITION
   STEP "Back Pos 1":   // S8
      // Move Position 1
              N    #"Move Position 1"
   END_STEP
   TRANSITION "Confirmation Pos 1" FROM "Back Pos 1" TO "Count Products"   // T7, jump: Conf Pos 1
      := #"Confimation Position 1";
   END_TRANSITION
   TRANSITION "Conf Side" FROM "Back Pos 1" TO "End Program"   // T8
      := #"Confimation Position 1";
   END_TRANSITION
   STEP "End Program":   // S9
   END_STEP
   TRANSITION "Products_ Zero" FROM "End Program" TO "Stop all axis"   // T9
      := #"Products zero";
   END_TRANSITION
   STEP "Stop all axis":   // S10
      // Reset Axis
              R    "Drive_1_Auto"
              R    "Drive_2_Auto"
              R    "PositionManagement".Demo_Pos.Start
   END_STEP
   TRANSITION True FROM "Stop all axis" TO Init   // T10, jump
      := TRUE;
   END_TRANSITION
END_FUNCTION_BLOCK

FUNCTION "SiemensEnc" : Void   // FC15, STL
TITLE = Test Siemens ENCODER
VERSION : 0.1
// stored: AutoNumber true, UDAEnableTagReadback false
BEGIN

NETWORK
TITLE = Presettings
      L     0;  //Delete control bits
      T     %DB1.DBD0;
      T     %DB1.DBD4;
      SET;
      S     %DB1.DBX4.0;  //Open SW gate









NETWORK
TITLE = Write to the control interface

NETWORK
TITLE = Read from the feedback interface
//Read 8 bytes from the 1 Count24V
//Configured start address of inputs
      L     "Tag_25":P;
      T     %DB1.DBD8;
      L     "Tag_26":P;
      T     %DB1.DBD12;
      R     %DB1.DBX4.0;  //Close SW gate



END_FUNCTION

FUNCTION "Axis_Confirmation" : Void   // FC7, FBD
TITLE = Axis Confirmation Block
VERSION : 0.1
// stored: AutoNumber true, IsIECCheckEnabled false, UDAEnableTagReadback false
   VAR_INPUT
      "Set Position" : Real;
   END_VAR
   VAR_OUTPUT
      "Axis On Position" : Bool;
      Min_Position_1 : Real;
      Max_Position_1 : Real;
   END_VAR
BEGIN

REGION Network 2: Calculate Position Tolerance 1
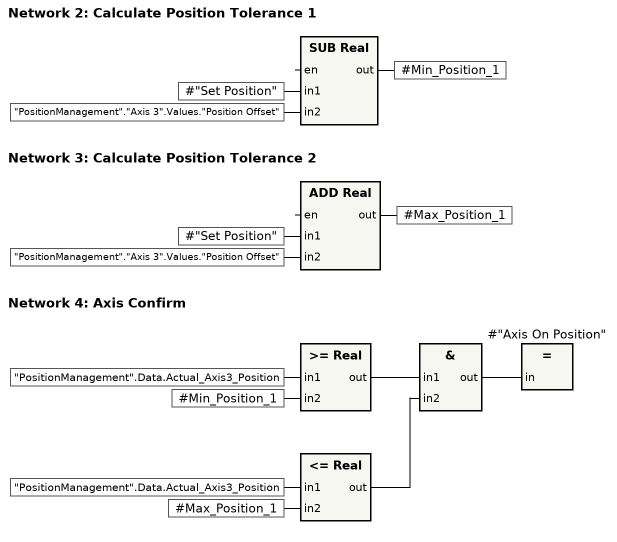
   #Min_Position_1 := #"Set Position" - "PositionManagement"."Axis 3".Values."Position Offset";
END_REGION

REGION Network 3: Calculate Position Tolerance 2
   #Max_Position_1 := #"Set Position" + "PositionManagement"."Axis 3".Values."Position Offset";
END_REGION

REGION Network 4: Axis Confirm
   #"Axis On Position" := ("PositionManagement".Data.Actual_Axis3_Position >= #Min_Position_1) AND ("PositionManagement".Data.Actual_Axis3_Position <= #Max_Position_1);
END_REGION
END_FUNCTION

FUNCTION_BLOCK "FB_EncoderFeedback_Degree"   // FB19, FBD
VERSION : 0.1
// stored: AutoNumber true, IsIECCheckEnabled false, UDAEnableTagReadback false
   VAR_INPUT
      CounterTag { ExternalVisible := 'False'; ExternalWritable := 'False'} : Int;   // Connect to the CounterTag IW102
      Position_Offset { ExternalVisible := 'False'; ExternalWritable := 'False'} : Real;   // Fill in the tolerance, when the axis approves the position. Above or below the desired position
      Pulsfactor { ExternalVisible := 'False'; ExternalWritable := 'False'} : Real;   // Number of pulses after 360 degree turn of the axis.
      Position_Correction { ExternalVisible := 'False'; ExternalWritable := 'False'} : Real;   // Small Position Correction for the Axis
      ReferenceRun_Command { ExternalVisible := 'False'; ExternalWritable := 'False'} : Bool;   // Command of starting the referencerun
      ReferenceSwitch { ExternalVisible := 'False'; ExternalWritable := 'False'} : Bool;   // ReferenceSwitch Mounted on Axis
      ReferencePosition { ExternalVisible := 'False'; ExternalWritable := 'False'} : Int;   // Position where the index puls of the reference switch enters.
   END_VAR
   VAR_OUTPUT
      Scaled_Position { ExternalVisible := 'False'; ExternalWritable := 'False'} : Real;   // Scaled Position scaled with Pulsfactor
      Actual_Enc_Pos { ExternalVisible := 'False'; ExternalWritable := 'False'} : Real;   // Actual Encoder Position
      AxisDB_Connection { ExternalVisible := 'False'; ExternalWritable := 'False'} : Real;   // Connection with Axis DB connection
   END_VAR
   VAR_TEMP
      Corrected_Axis_Pos : Real;
      Unscaled_Position : Int;   // Unscaled Position of the Encoder
      Unsc2 : Int;   // Unsc 2 position
      Act_Enc_Pos_Int : DInt;
      Scaled_Position_Real : Real;
      PosDint : DInt;
      Unscaled_Position_Real : Real;
      InternalCounter : Int;
      CalDifCounter : Int;
      Pos_Storage : Int;
      Pos_Diffrence : Int;
      Add_Pos : Int;
      Sub_Pos : Int;
      LessThanZero : Bool;
      LTZ_out : Int;
   END_VAR
BEGIN

REGION Network 2: SPARE
END_REGION

NETWORK
TITLE = Call the Countermodule
      L     #CounterTag;  //Van tellerkaart TAG Gelinkt aan IW102
      L     "PositionManagement".Data.CntPlsPrev;  //Vorige scan
      -D;
      T     "PositionManagement".Data.CntPlsDiff;  //Verschil

      L     "PositionManagement".Data.CntPlsDiff;  // Verschil groter dan nul?
      L     0;
      >D;
      JCN   chkneg;

      L     "PositionManagement".Data.CntPlsDiff;  //Verschil optellen bij actuele pulswaarde
      L     "PositionManagement".Data.CntPlsAct;
      +D;
      T     "PositionManagement".Data.CntPlsAct;
      JU    end;  //rest overslaan.

chkneg:L     "PositionManagement".Data.CntPlsDiff;  // Verschil groter dan nul?
      L     0;
      <D;
      JCN   end;
      L     -1;  //verschil positief maken
      *D;
      T     "PositionManagement".Data.CntPlsDiff;  //verschil positief

      L     "PositionManagement".Data.CntPlsAct;  //Verschil optellen bij actuele pulswaarde
      +D;
      T     "PositionManagement".Data.CntPlsAct;

end:  NOP   0;

      L     #CounterTag;
      T     "PositionManagement".Data.CntPlsPrev;


REGION Network 4: Store Old Position
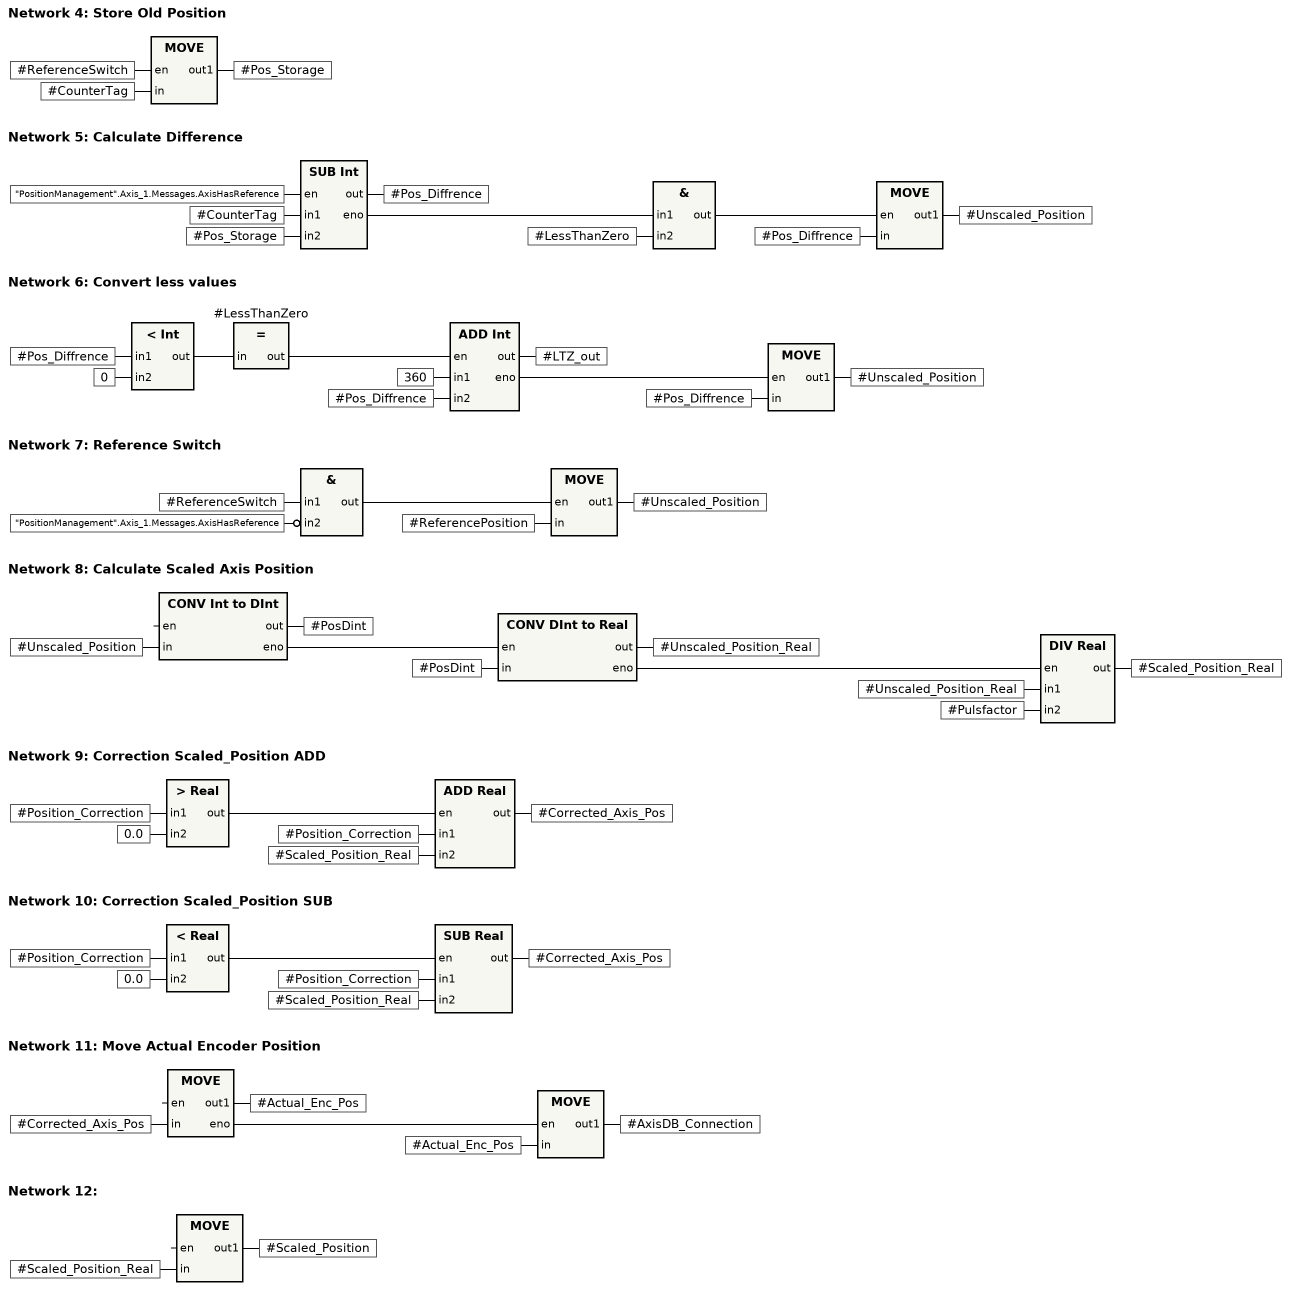
   IF #ReferenceSwitch THEN #Pos_Storage := #CounterTag; END_IF;
END_REGION

REGION Network 5: Calculate Difference
   // ENO of a box is taken as its EN; it also drops when the box reports an error
   IF "PositionManagement".Axis_1.Messages.AxisHasReference THEN
       #Pos_Diffrence := #CounterTag - #Pos_Storage;
   END_IF;
   IF "PositionManagement".Axis_1.Messages.AxisHasReference AND #LessThanZero THEN
       #Unscaled_Position := #Pos_Diffrence;
   END_IF;
END_REGION

REGION Network 6: Convert less values
   // ENO of a box is taken as its EN; it also drops when the box reports an error
   #LessThanZero := #Pos_Diffrence < 0;
   IF #LessThanZero THEN
       #LTZ_out := 360 + #Pos_Diffrence;
       #Unscaled_Position := #Pos_Diffrence;
   END_IF;
END_REGION

REGION Network 7: Reference Switch
   IF #ReferenceSwitch AND NOT "PositionManagement".Axis_1.Messages.AxisHasReference THEN
       #Unscaled_Position := #ReferencePosition;
   END_IF;
END_REGION

REGION Network 8: Calculate Scaled Axis Position
   // ENO of a box is taken as its EN; it also drops when the box reports an error
   #PosDint := INT_TO_DINT(#Unscaled_Position);
   #Unscaled_Position_Real := DINT_TO_REAL(#PosDint);
   #Scaled_Position_Real := #Unscaled_Position_Real / #Pulsfactor;
END_REGION

REGION Network 9: Correction Scaled_Position ADD
   IF #Position_Correction > 0.0 THEN
       #Corrected_Axis_Pos := #Position_Correction + #Scaled_Position_Real;
   END_IF;
END_REGION

REGION Network 10: Correction Scaled_Position SUB
   IF #Position_Correction < 0.0 THEN
       #Corrected_Axis_Pos := #Position_Correction - #Scaled_Position_Real;
   END_IF;
END_REGION

REGION Network 11: Move Actual Encoder Position
   // ENO of a box is taken as its EN; it also drops when the box reports an error
   #Actual_Enc_Pos := #Corrected_Axis_Pos;
   #AxisDB_Connection := #Actual_Enc_Pos;
END_REGION

REGION Network 12
   #Scaled_Position := #Scaled_Position_Real;
END_REGION
END_FUNCTION_BLOCK

FUNCTION "StartInfeedBelt_FBD" : Void   // FC11, FBD
TITLE = StartInfeedBelt
VERSION : 0.1
// stored: AutoNumber true, IsIECCheckEnabled false, UDAEnableTagReadback false
   VAR_INPUT
      SystemRun_Command : Bool;
   END_VAR
BEGIN

REGION Network 2: Aanvoerband (1) - Aansturen
   // This block sets an starttimer on Drive 1
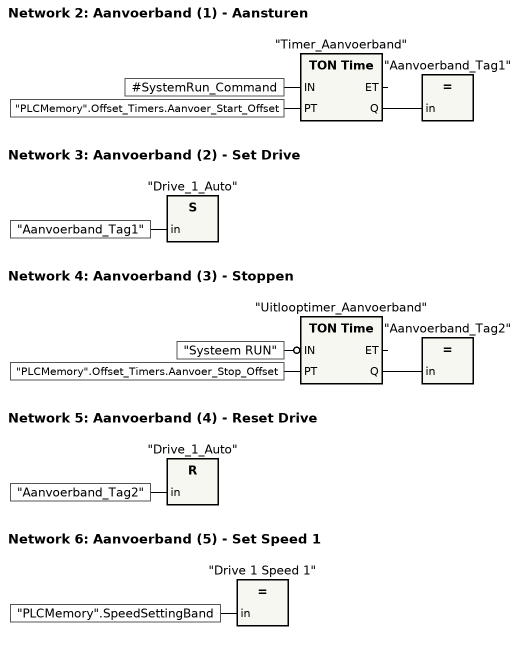
   "Timer_Aanvoerband".TON(IN := #SystemRun_Command, PT := "PLCMemory".Offset_Timers.Aanvoer_Start_Offset);
   "Aanvoerband_Tag1" := "Timer_Aanvoerband".Q;
END_REGION

REGION Network 3: Aanvoerband (2) - Set Drive
   // This block sets Drive 1 Auto signal
   IF "Aanvoerband_Tag1" THEN "Drive_1_Auto" := TRUE; END_IF;
END_REGION

REGION Network 4: Aanvoerband (3) - Stoppen
   // This block sets an End timer on Drive 1
   "Uitlooptimer_Aanvoerband".TON(IN := NOT "Systeem RUN", PT := "PLCMemory".Offset_Timers.Aanvoer_Stop_Offset);
   "Aanvoerband_Tag2" := "Uitlooptimer_Aanvoerband".Q;
END_REGION

REGION Network 5: Aanvoerband (4) - Reset Drive
   // This block resets Drive 1 Auto
   IF "Aanvoerband_Tag2" THEN "Drive_1_Auto" := FALSE; END_IF;
END_REGION

REGION Network 6: Aanvoerband (5) - Set Speed 1
   // This block sets the speed for Drive 1
   "Drive 1 Speed 1" := "PLCMemory".SpeedSettingBand;
END_REGION
END_FUNCTION

FUNCTION_BLOCK "TestingAndOld"   // FB24, LAD
VERSION : 0.1
// stored: AutoNumber true, IsIECCheckEnabled false, UDAEnableTagReadback false
   VAR_TEMP
      NotUsed : Bool;
      SAFE_OK_Signal : Bool;
      ScPos : Real;
      ActEncPos : Real;
      DB : Real;
   END_VAR
BEGIN

REGION Network 2: Encoder Feedback Connection FB
   // Getting the feedback from the encoder device
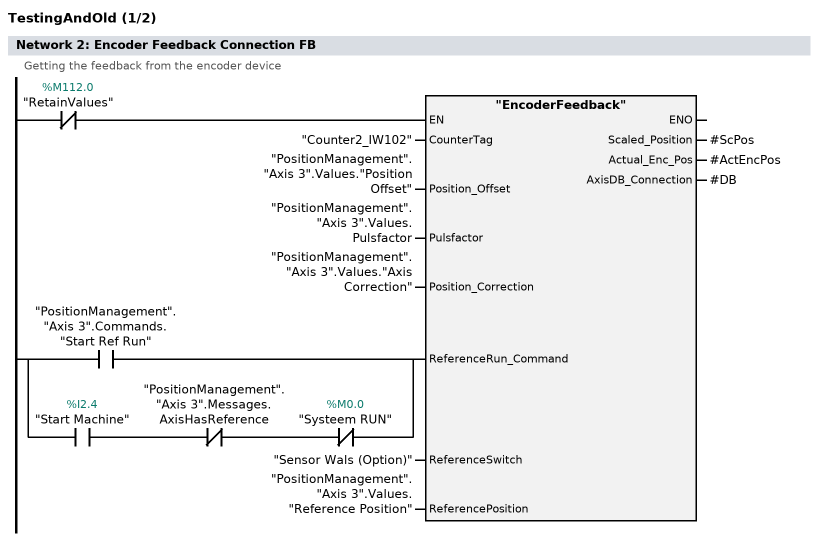
   RUNG wire#powerrail
      I_Contact( "RetainValues" )
      "EncoderFeedback"(ReferenceRun_Command := wire#w1, CounterTag := "Counter2_IW102", Position_Offset := "PositionManagement"."Axis 3".Values."Position Offset", Pulsfactor := "PositionManagement"."Axis 3".Values.Pulsfactor, Position_Correction := "PositionManagement"."Axis 3".Values."Axis Correction", ReferenceSwitch := "Sensor Wals (Option)", ReferencePosition := "PositionManagement"."Axis 3".Values."Reference Position", Scaled_Position => #ScPos, Actual_Enc_Pos => #ActEncPos, AxisDB_Connection => #DB)
   END_RUNG
   RUNG wire#powerrail
      Contact( "PositionManagement"."Axis 3".Commands."Start Ref Run" )
   END_RUNG wire#w1
   RUNG wire#powerrail
      Contact( "Start Machine" )
      I_Contact( "PositionManagement"."Axis 3".Messages.AxisHasReference )
      I_Contact( "Systeem RUN" )
   END_RUNG wire#w1
   // the same network as SCL:
   IF NOT "RetainValues" THEN
       "EncoderFeedback"(CounterTag := "Counter2_IW102",
                         Position_Offset := "PositionManagement"."Axis 3".Values."Position Offset",
                         Pulsfactor := "PositionManagement"."Axis 3".Values.Pulsfactor,
                         Position_Correction := "PositionManagement"."Axis 3".Values."Axis Correction",
                         ReferenceRun_Command := "PositionManagement"."Axis 3".Commands."Start Ref Run" OR ("Start Machine" AND NOT "PositionManagement"."Axis 3".Messages.AxisHasReference AND NOT "Systeem RUN"),
                         ReferenceSwitch := "Sensor Wals (Option)",
                         ReferencePosition := "PositionManagement"."Axis 3".Values."Reference Position",
                         Scaled_Position => #ScPos,
                         Actual_Enc_Pos => #ActEncPos,
                         AxisDB_Connection => #DB);
   END_IF;
END_REGION

REGION Network 3: Drive Manager Axis 3
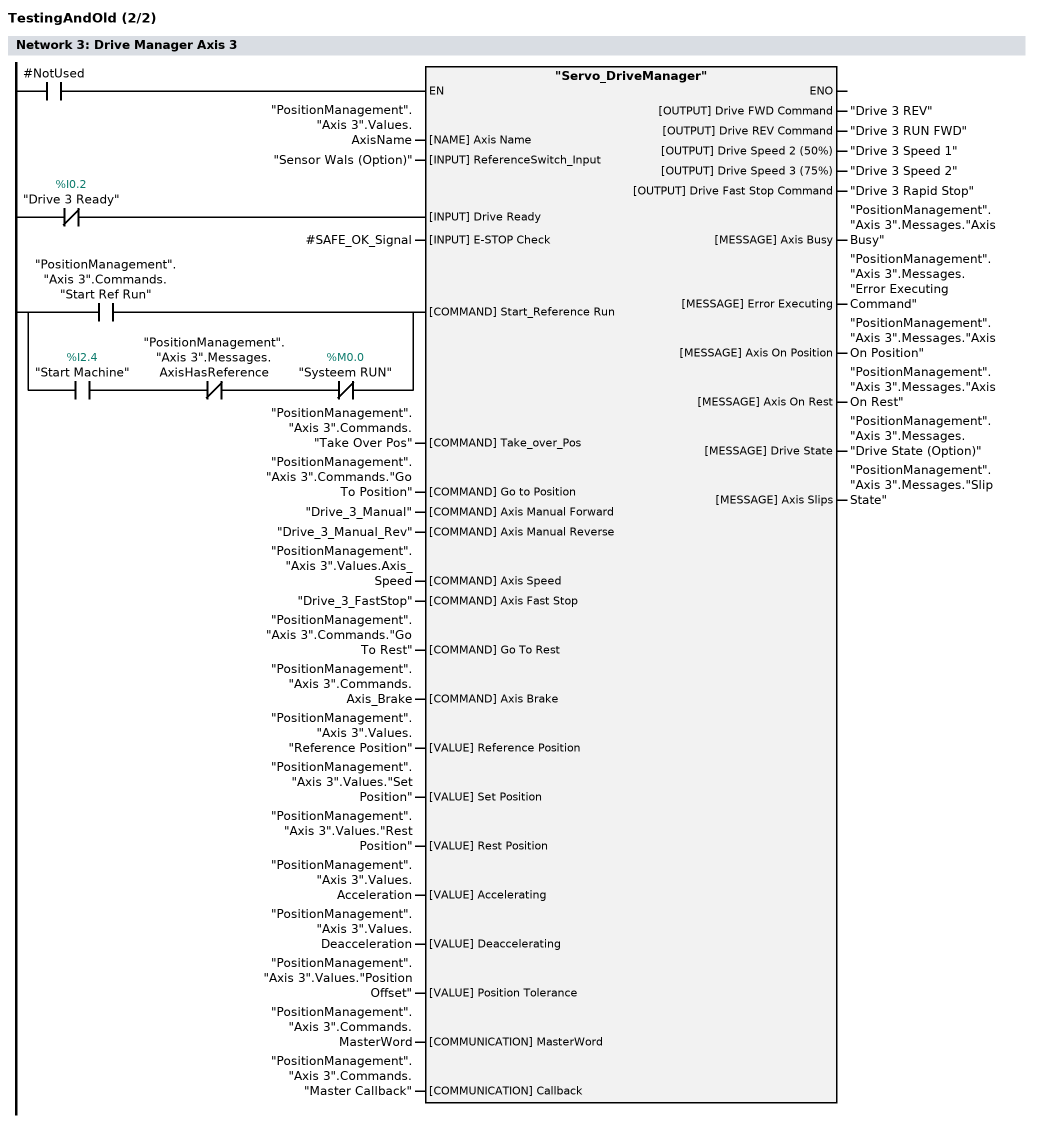
   RUNG wire#powerrail
      Contact( #NotUsed )
      "Servo_DriveManager"("[INPUT] Drive Ready" := wire#w1, "[COMMAND] Start_Reference Run" := wire#w2, "[NAME] Axis Name" := "PositionManagement"."Axis 3".Values.AxisName, "[INPUT] ReferenceSwitch_Input" := "Sensor Wals (Option)", "[INPUT] E-STOP Check" := #SAFE_OK_Signal, "[COMMAND] Take_over_Pos" := "PositionManagement"."Axis 3".Commands."Take Over Pos", "[COMMAND] Go to Position" := "PositionManagement"."Axis 3".Commands."Go To Position", "[COMMAND] Axis Manual Forward" := "Drive_3_Manual", "[COMMAND] Axis Manual Reverse" := "Drive_3_Manual_Rev", "[COMMAND] Axis Speed" := "PositionManagement"."Axis 3".Values.Axis_Speed, "[COMMAND] Axis Fast Stop" := "Drive_3_FastStop", "[COMMAND] Go To Rest" := "PositionManagement"."Axis 3".Commands."Go To Rest", "[COMMAND] Axis Brake" := "PositionManagement"."Axis 3".Commands.Axis_Brake, "[VALUE] Reference Position" := "PositionManagement"."Axis 3".Values."Reference Position", "[VALUE] Set Position" := "PositionManagement"."Axis 3".Values."Set Position", "[VALUE] Rest Position" := "PositionManagement"."Axis 3".Values."Rest Position", "[VALUE] Accelerating" := "PositionManagement"."Axis 3".Values.Acceleration, "[VALUE] Deaccelerating" := "PositionManagement"."Axis 3".Values.Deacceleration, "[VALUE] Position Tolerance" := "PositionManagement"."Axis 3".Values."Position Offset", "[COMMUNICATION] MasterWord" := "PositionManagement"."Axis 3".Commands.MasterWord, "[COMMUNICATION] Callback" := "PositionManagement"."Axis 3".Commands."Master Callback", "[OUTPUT] Drive FWD Command" => "Drive 3 REV", "[OUTPUT] Drive REV Command" => "Drive 3 RUN FWD", "[OUTPUT] Drive Speed 2 (50%)" => "Drive 3 Speed 1", "[OUTPUT] Drive Speed 3 (75%)" => "Drive 3 Speed 2", "[OUTPUT] Drive Fast Stop Command" => "Drive 3 Rapid Stop", "[MESSAGE] Axis Busy" => "PositionManagement"."Axis 3".Messages."Axis Busy", "[MESSAGE] Error Executing" => "PositionManagement"."Axis 3".Messages."Error Executing Command", "[MESSAGE] Axis On Position" => "PositionManagement"."Axis 3".Messages."Axis On Position", "[MESSAGE] Axis On Rest" => "PositionManagement"."Axis 3".Messages."Axis On Rest", "[MESSAGE] Drive State" => "PositionManagement"."Axis 3".Messages."Drive State (Option)", "[MESSAGE] Axis Slips" => "PositionManagement"."Axis 3".Messages."Slip State")
   END_RUNG
   RUNG wire#powerrail
      I_Contact( "Drive 3 Ready" )
   END_RUNG wire#w1
   RUNG wire#powerrail
      Contact( "PositionManagement"."Axis 3".Commands."Start Ref Run" )
   END_RUNG wire#w2
   RUNG wire#powerrail
      Contact( "Start Machine" )
      I_Contact( "PositionManagement"."Axis 3".Messages.AxisHasReference )
      I_Contact( "Systeem RUN" )
   END_RUNG wire#w2
   // the same network as SCL:
   IF #NotUsed THEN
       "Servo_DriveManager"("[NAME] Axis Name" := "PositionManagement"."Axis 3".Values.AxisName,
                            "[INPUT] ReferenceSwitch_Input" := "Sensor Wals (Option)",
                            "[INPUT] Drive Ready" := NOT "Drive 3 Ready",
                            "[INPUT] E-STOP Check" := #SAFE_OK_Signal,
                            "[COMMAND] Start_Reference Run" := "PositionManagement"."Axis 3".Commands."Start Ref Run" OR ("Start Machine" AND NOT "PositionManagement"."Axis 3".Messages.AxisHasReference AND NOT "Systeem RUN"),
                            "[COMMAND] Take_over_Pos" := "PositionManagement"."Axis 3".Commands."Take Over Pos",
                            "[COMMAND] Go to Position" := "PositionManagement"."Axis 3".Commands."Go To Position",
                            "[COMMAND] Axis Manual Forward" := "Drive_3_Manual",
                            "[COMMAND] Axis Manual Reverse" := "Drive_3_Manual_Rev",
                            "[COMMAND] Axis Speed" := "PositionManagement"."Axis 3".Values.Axis_Speed,
                            "[COMMAND] Axis Fast Stop" := "Drive_3_FastStop",
                            "[COMMAND] Go To Rest" := "PositionManagement"."Axis 3".Commands."Go To Rest",
                            "[COMMAND] Axis Brake" := "PositionManagement"."Axis 3".Commands.Axis_Brake,
                            "[VALUE] Reference Position" := "PositionManagement"."Axis 3".Values."Reference Position",
                            "[VALUE] Set Position" := "PositionManagement"."Axis 3".Values."Set Position",
                            "[VALUE] Rest Position" := "PositionManagement"."Axis 3".Values."Rest Position",
                            "[VALUE] Accelerating" := "PositionManagement"."Axis 3".Values.Acceleration,
                            "[VALUE] Deaccelerating" := "PositionManagement"."Axis 3".Values.Deacceleration,
                            "[VALUE] Position Tolerance" := "PositionManagement"."Axis 3".Values."Position Offset",
                            "[COMMUNICATION] MasterWord" := "PositionManagement"."Axis 3".Commands.MasterWord,
                            "[COMMUNICATION] Callback" := "PositionManagement"."Axis 3".Commands."Master Callback",
                            "[OUTPUT] Drive FWD Command" => "Drive 3 REV",
                            "[OUTPUT] Drive REV Command" => "Drive 3 RUN FWD",
                            "[OUTPUT] Drive Speed 2 (50%)" => "Drive 3 Speed 1",
                            "[OUTPUT] Drive Speed 3 (75%)" => "Drive 3 Speed 2",
                            "[OUTPUT] Drive Fast Stop Command" => "Drive 3 Rapid Stop",
                            "[MESSAGE] Axis Busy" => "PositionManagement"."Axis 3".Messages."Axis Busy",
                            "[MESSAGE] Error Executing" => "PositionManagement"."Axis 3".Messages."Error Executing Command",
                            "[MESSAGE] Axis On Position" => "PositionManagement"."Axis 3".Messages."Axis On Position",
                            "[MESSAGE] Axis On Rest" => "PositionManagement"."Axis 3".Messages."Axis On Rest",
                            "[MESSAGE] Drive State" => "PositionManagement"."Axis 3".Messages."Drive State (Option)",
                            "[MESSAGE] Axis Slips" => "PositionManagement"."Axis 3".Messages."Slip State");
   END_IF;
END_REGION
END_FUNCTION_BLOCK

FUNCTION_BLOCK "SCLTestingEnc"
{ S7_Optimized_Access := 'FALSE' }
VERSION : 0.1
   VAR_TEMP 
      tempDWord : Word;
      LocalCtrlWord : Word;
      CtrlWordDword : DWord;
      WordLow : Word;
      WordHigh : Word;
      InLow : Word;
      InHigh : Word;
      RawDINT : DInt;
      TempControl : DWord;
   END_VAR


BEGIN
	// --- ControlWord opbouwen (gate openen via bit 0)
	IF "DB_EncoderBand".EnableGate THEN
	    "DB_EncoderBand".ControlWord := 16#0001; // Alleen bit 0 actief
	ELSE
	    "DB_EncoderBand".ControlWord := 16#0000;
	END_IF;
	
	// --- Omzetten naar DWORD
	#CtrlWordDword := WORD_TO_DWORD("DB_EncoderBand".ControlWord);
	
	// --- Opsplitsen in 2 WORDs
	#WordLow := DWORD_TO_WORD(#CtrlWordDword AND 16#0000FFFF);
	#WordHigh := DWORD_TO_WORD(DWORD_TO_DINT(#CtrlWordDword) / 65536);
	
	// --- Wegschrijven naar uitgangsgebied (1Count kaart op QW110/QW112)
	"Enable" := #WordLow;
	"Tag_61" := #WordHigh;
	
	// --- Inlezen uit 1Count kaart (IW110/IW112)
	#InLow := "EncoderBand_Alive";
	#InHigh := "Enc3(6)";
	
	// --- Samenvoegen tot DINT
	#RawDINT := WORD_TO_DINT(#InLow) + (WORD_TO_DINT(#InHigh) * 65536);
	
	// --- Wegschrijven naar datablock
	"DB_EncoderBand".EncoderValue := #RawDINT;
	
	//Enable Word
	"DB_EncoderBand".ControlWord := 16#0041; // Bit 6 + Bit 0 (sommige kaarten vereisen extra enable-bits)
	
	
END_FUNCTION_BLOCK

FUNCTION_BLOCK "FB_ProductTrigger"
{ S7_Optimized_Access := 'FALSE' }
VERSION : 0.1
   VAR_INPUT 
      SensorInput : Bool;
      TimeDelay : Time;
      SystemTime : Time;
   END_VAR

   VAR_OUTPUT 
      TriggerMovement : Bool;
      ProductCount : Int;
   END_VAR

   VAR_TEMP 
      ProductQueue : Array[0..1] of "ProductEntry";
      SensorMemory : Bool;
      i : Int;
   END_VAR


BEGIN
	// Reset output
	#TriggerMovement := FALSE;
	
	// Flankdetectie op sensor
	IF #SensorInput AND NOT #SensorMemory THEN
	    // Zoek eerste vrije plek
	    FOR #i := 1 TO 10 DO
	        IF NOT #ProductQueue[#i].Active THEN
	            #ProductQueue[#i].Active := TRUE;
	            #ProductQueue[#i].StartTime := #SystemTime;
	            EXIT;
	        END_IF;
	    END_FOR;
	END_IF;
	#SensorMemory := #SensorInput;
	
	// Kijk of een van de producten klaar is voor beweging
	FOR #i := 1 TO 10 DO
	    IF #ProductQueue[#i].Active AND (#SystemTime - #ProductQueue[#i].StartTime >= #TimeDelay) THEN
	        #TriggerMovement := TRUE;
	        #ProductQueue[#i].Active := FALSE; // Verwijder uit wachtrij
	        EXIT; // Eén tegelijk
	    END_IF;
	END_FOR;
	
	// Update productenteller
	#ProductCount := 0;
	FOR #i := 1 TO 10 DO
	    IF #ProductQueue[#i].Active THEN
	        #ProductCount := #ProductCount + 1;
	    END_IF;
	END_FOR;
	
END_FUNCTION_BLOCK

FUNCTION_BLOCK "FB_SystemTimeCounter"
{ S7_Optimized_Access := 'FALSE' }
VERSION : 0.1
   VAR_INPUT 
      Enable : Bool;
      CycleTime : Time;
   END_VAR

   VAR_OUTPUT 
      SystemTime : Time;
   END_VAR

   VAR_TEMP 
      PrevEnable : Bool;
   END_VAR


BEGIN
	//Start//
	
	IF #Enable THEN
	    // Enkel verhogen als Enable TRUE is
	    #SystemTime := #SystemTime + #CycleTime;
	END_IF;
	
	// Reset eventueel bij FALSE->TRUE flank
	//IF NOT #PrevEnable AND #Enable THEN
	    // Optioneel reset: SystemTime := T#0s;
	//END_IF;
	
	#PrevEnable := #Enable;
	
	
	
END_FUNCTION_BLOCK

FUNCTION "Servo360Axis" : Void
{ S7_Optimized_Access := 'FALSE' }
VERSION : 0.1
   VAR_INPUT 
      ActEncPos : Real;
      "[NAME] Axis Name" : String;
      "[INPUT] ReferenceSwitch_Input" : Bool;
      "[INPUT] Drive Ready" : Bool;
      "[INPUT] E-STOP Check" : Bool;
      "[COMMAND] Start_Reference Run" : Bool;
      "[COMMAND] Take_over_Pos" : Bool;
      "[COMMAND] Go to Position" : Bool;
      "[COMMAND] Axis Manual Forward" : Bool;
      "[COMMAND] Axis Manual Reverse" : Bool;
      "[COMMAND] Axis Speed" : Int;
      "[COMMAND] Axis Fast Stop" : Bool;
      "[COMMAND] Go To Rest" : Bool;
      "[COMMAND] Axis Brake" : Bool;
      "[VALUE] Reference Position" : Int;
      "[VALUE] Set Position" : Real;
      "[VALUE] Rest Position" : Real;
      "[VALUE] Accelerating" : Real;
      "[VALUE] Deaccelerating" : Real;
      "[VALUE] Position Tolerance" : Real;
      "[VALUE] Modulo Factor" : Real;
      "[COMMUNICATION] MasterWord" : String;
      "[COMMUNICATION] Callback" : String;
      "[VALUE] Pulsfactor" : Int;
   END_VAR

   VAR_OUTPUT 
      "[OUTPUT] Drive FWD Command" : Bool;
      "[OUTPUT] Drive REV Command" : Bool;
      "[OUTPUT] Drive Speed 2 (50%)" : Bool;
      "[OUTPUT] Drive Speed 3 (75%)" : Bool;
      "[OUTPUT] Drive Fast Stop Command" : Bool;
      "[MESSAGE] Axis Busy" : Bool;
      "[MESSAGE] Error Executing" : Bool;
      "[MESSAGE] Axis On Position" : Bool;
      "[MESSAGE] Axis On Rest" : Bool;
      "[MESSAGE] Drive State" : String;
      "[MESSAGE] Axis Slips" : String;
   END_VAR

   VAR_TEMP 
      UnscPos : Bool;
      ScPos : Bool;
      SetRefRun : Bool;
      SetRefRun_Q : Bool;
      MoveToRest : Bool;
      MoveToRest_Q : Bool;
      Automatic_Positive : Bool;
      Manual_Positive : Bool;
      Automatic_Negative : Bool;
      Manual_Negative : Bool;
      HS_Positive : Bool;
      MasterWordHex : Bool;
      Speed50 : Bool;
      Speed75 : Bool;
      Min_Position : Real;
      Max_Position : Real;
      Axis_On_Position : Bool;
      Direction_Forward : Bool;
      Direction_Backward : Bool;
      Drive_Auto_Fwd : Bool;
      InternalFastStop : Bool;
      RefRunSetSignal : Bool;
      GoToRest2 : Bool;
      "[COMMAND] Go to Position_Rest" : Bool;
      RestPos_SpareMove : Bool;
      tmp : Real;
      diff : Real;
      AbsDiff : Real;
      HalfModulo : Real;
      TargetPos : Real;
      RefTarget : Real;
      RefDiff : Real;
      RefAbs : Real;
      RefBusy : Bool;
      RefMode : Bool;
      AutoMode : Bool;
      ActiveTarget : Real;
      DirCmd : Int;
      AbsDiffActive : Real;
      TolStop : Real;
      TolSwitch : Real;
      diffActive : Real;
      RefSw_Old : Bool;
      "[VALUE] Position Offset" : Int;
      _ppu : Int;
      AutoMove_Q : Bool;
      GoPos_Old : Bool;
   END_VAR


BEGIN
	// =======================
	// ====== IMPLEMENT ======
	// =======================
	
	// --- 0. Safety (fast stop)
	#"[OUTPUT] Drive Fast Stop Command" := #"[COMMAND] Axis Fast Stop" OR (NOT #"[INPUT] E-STOP Check");
	
	// --- 1. Referentie-latch (SR)
	IF #"[INPUT] ReferenceSwitch_Input" THEN
	    #"SetRefRun_Q" := FALSE; // switch geraakt -> referentie klaar
	ELSIF #"[COMMAND] Start_Reference Run" THEN
	    #"SetRefRun_Q" := TRUE;  // start ref
	END_IF;
	
	// --- 2. GoTo latch (pulsbestendig)
	IF (NOT #"GoPos_Old") AND #"[COMMAND] Go to Position" AND #"[INPUT] Drive Ready" AND #"[INPUT] E-STOP Check" THEN
	    #"AutoMove_Q" := TRUE;
	END_IF;
	#"GoPos_Old" := #"[COMMAND] Go to Position";
	
	// --- 3. Modus (exclusief: Ref heeft voorrang)
	#"RefMode" := #"SetRefRun_Q" AND (NOT #"[INPUT] ReferenceSwitch_Input");
	
	// Auto actief zolang gelatcht, mits niet in Ref
	
	    // reset automove bij aankomen of door safety/fast stop
	    IF #"[OUTPUT] Drive Fast Stop Command" OR (NOT #"[INPUT] Drive Ready") OR (NOT #"[INPUT] E-STOP Check") THEN
	        #"AutoMove_Q" := FALSE;
	    END_IF;
	
	
	
	#_ppu := #"[VALUE] Pulsfactor";
	IF #_ppu <= 0.0 THEN
	    #_ppu := 1; // anti-div/0
	END_IF;
	
	#"ActEncPos" := INT_TO_REAL("Counter2_IW102") / #_ppu + #"[VALUE] Position Offset";
	
	// --- 5. Active target
	IF #"RefMode" THEN
	    #"ActiveTarget" := INT_TO_REAL(#"[VALUE] Reference Position");
	ELSE
	    #"ActiveTarget" := #"[VALUE] Set Position";
	END_IF;
	
	// --- 6. Diff + modulo (kortste pad)
	#"diff" := #"ActiveTarget" - #"ActEncPos";
	
	IF #"[VALUE] Modulo Factor" > 0.0 THEN
	    // normaliseer (-Modulo .. +Modulo)
	    WHILE #"diff" >= #"[VALUE] Modulo Factor" DO
	        #"diff" := #"diff" - #"[VALUE] Modulo Factor";
	    END_WHILE;
	    WHILE #"diff" < - #"[VALUE] Modulo Factor" DO
	        #"diff" := #"diff" + #"[VALUE] Modulo Factor";
	    END_WHILE;
	    
	    // kortste pad (± Modulo/2)
	    IF #"diff" > (#"[VALUE] Modulo Factor" * 0.5) THEN
	        #"diff" := #"diff" - #"[VALUE] Modulo Factor";
	    ELSIF #"diff" < - (#"[VALUE] Modulo Factor" * 0.5) THEN
	        #"diff" := #"diff" + #"[VALUE] Modulo Factor";
	    END_IF;
	END_IF;
	
	#"AbsDiff" := ABS(#"diff");
	
	// --- 7. Hysterese-banden
	#"TolStop" := #"[VALUE] Position Tolerance";
	IF #"TolStop" < 0.0 THEN
	    #"TolStop" := 0.0;
	END_IF;
	
	// "TolSwitch" = max(1.5*TolStop, TolStop+0.01)  → zonder MAX()
	#"TolSwitch" := #"TolStop" * 1.5;
	IF (#"TolStop" + 0.01) > #"TolSwitch" THEN
	    #"TolSwitch" := #"TolStop" + 0.01;
	END_IF;
	
	// --- 8. OnPosition (alleen betekenisvol in Auto)
	IF #"RefMode" THEN
	    #"[MESSAGE] Axis On Position" := FALSE;
	ELSE
	    #"[MESSAGE] Axis On Position" := (#"AbsDiff" <= #"TolStop");
	    // AutoMove reset bij aankomen
	    IF #"[MESSAGE] Axis On Position" THEN
	        #"AutoMove_Q" := FALSE;
	    END_IF;
	END_IF;
	
	// --- 9. Manual overrides (niet tijdens ref)
	#"Manual_Positive" := (NOT #"RefMode") AND #"[COMMAND] Axis Manual Forward" AND NOT #"[COMMAND] Axis Manual Reverse";
	#"Manual_Negative" := (NOT #"RefMode") AND #"[COMMAND] Axis Manual Reverse" AND NOT #"[COMMAND] Axis Manual Forward";
	
	// --- 10. Busy (ref of automove of manual) + safety
	#"[MESSAGE] Axis Busy" :=
	(
	(#"RefMode" OR #"AutoMove_Q" OR #"Manual_Positive" OR #"Manual_Negative")
	AND #"[INPUT] Drive Ready"
	AND #"[INPUT] E-STOP Check"
	);
	
	// --- 11. Richting met hysterese (op basis van Diff)
	IF #"AbsDiff" <= #"TolStop" THEN
	    #"DirCmd" := 0; // STOP
	ELSIF #"AbsDiff" >= #"TolSwitch" THEN
	    IF #"diff" > 0.0 THEN
	        #"DirCmd" := 1;  // FWD
	    ELSIF #"diff" < 0.0 THEN
	        #"DirCmd" := -1; // REV
	    END_IF;
	END_IF;
	
	
	
	// --- 12. Speed select (minstens één speed aan tijdens bewegen)
	#"[OUTPUT] Drive Speed 2 (50%)" := FALSE;
	#"[OUTPUT] Drive Speed 3 (75%)" := FALSE;
	
	IF #"[MESSAGE] Axis Busy" THEN
	    IF #"[COMMAND] Axis Speed" >= 75 THEN
	        #"[OUTPUT] Drive Speed 3 (75%)" := TRUE;
	    ELSE
	        #"[OUTPUT] Drive Speed 2 (50%)" := TRUE; // default
	    END_IF;
	END_IF;
	
	// --- 13. Outputs (prioriteit: Manual > Ref/Auto; alleen bij Busy & safety)
	#"[OUTPUT] Drive FWD Command" := FALSE;
	#"[OUTPUT] Drive REV Command" := FALSE;
	
	IF #"[INPUT] Drive Ready" AND #"[INPUT] E-STOP Check" AND #"[MESSAGE] Axis Busy" THEN
	    // Manual
	    IF #"Manual_Positive" THEN
	        #"[OUTPUT] Drive FWD Command" := TRUE;
	    ELSIF #"Manual_Negative" THEN
	        #"[OUTPUT] Drive REV Command" := TRUE;
	    ELSE
	        // Ref/Auto
	        CASE #"DirCmd" OF
	            1:
	                #"[OUTPUT] Drive FWD Command" := TRUE;
	            -1:
	                #"[OUTPUT] Drive REV Command" := TRUE;
	        END_CASE;
	    END_IF;
	END_IF;
	
	// Safety en autostop bij bereikt (alleen in Auto)
	IF (NOT #"[INPUT] Drive Ready") OR (NOT #"[INPUT] E-STOP Check") OR ((NOT #"RefMode") AND #"[MESSAGE] Axis On Position") THEN
	    #"[OUTPUT] Drive FWD Command" := FALSE;
	    #"[OUTPUT] Drive REV Command" := FALSE;
	    // bij autostop ook speed uit
	    IF (NOT #"RefMode") AND #"[MESSAGE] Axis On Position" THEN
	        #"[OUTPUT] Drive Speed 2 (50%)" := FALSE;
	        #"[OUTPUT] Drive Speed 3 (75%)" := FALSE;
	    END_IF;
	END_IF;
	
	// --- 14. Referentie-offset zetten op flank van switch
	IF (NOT #"RefSw_Old") AND #"[INPUT] ReferenceSwitch_Input" THEN
	    // offset = RefPos - (raw/ppu)
	    #"[VALUE] Position Offset" := (#"[VALUE] Reference Position") - ("Counter2_IW102") / #_ppu;
	    #"SetRefRun_Q" := FALSE; // ref klaar
	END_IF;
	#"RefSw_Old" := #"[INPUT] ReferenceSwitch_Input";
	
	// --- 15. State string
	IF #"[OUTPUT] Drive Fast Stop Command" THEN
	    #"[MESSAGE] Drive State" := 'FAST STOP';
	ELSIF #"[OUTPUT] Drive FWD Command" THEN
	    IF #"[OUTPUT] Drive Speed 3 (75%)" THEN
	        #"[MESSAGE] Drive State" := 'RUN FWD / 75%';
	    ELSE
	        #"[MESSAGE] Drive State" := 'RUN FWD / 50%';
	    END_IF;
	ELSIF #"[OUTPUT] Drive REV Command" THEN
	    IF #"[OUTPUT] Drive Speed 3 (75%)" THEN
	        #"[MESSAGE] Drive State" := 'RUN REV / 75%';
	    ELSE
	        #"[MESSAGE] Drive State" := 'RUN REV / 50%';
	    END_IF;
	ELSE
	    IF #"RefMode" THEN
	        #"[MESSAGE] Drive State" := 'REF RUN';
	    ELSIF #"[MESSAGE] Axis On Position" THEN
	        #"[MESSAGE] Drive State" := 'ON POSITION';
	    ELSE
	        #"[MESSAGE] Drive State" := 'IDLE';
	    END_IF;
	END_IF;
	
END_FUNCTION

DATA_BLOCK "2in-1out_Block_Start_Stop_Override"   // DB6
VERSION : 0.1
// stored: AutoNumber true, InstanceOfName 2in-1out_Block, InstanceOfType FB
"2in-1out_Block"
BEGIN
END_DATA_BLOCK

DATA_BLOCK "ProductBuffer_V3_BehindWals_DB"   // DB2
VERSION : 0.1
// stored: AutoNumber true, InstanceOfName ProductBuffer_V3, InstanceOfType FB
"ProductBuffer_V3"
BEGIN
END_DATA_BLOCK

DATA_BLOCK "ProductBuffer_V3_DB"   // DB90
VERSION : 0.1
// stored: AutoNumber true, InstanceOfName ProductBuffer_V3, InstanceOfType FB
"ProductBuffer_V3"
BEGIN
END_DATA_BLOCK

DATA_BLOCK "SCLTestingEnc_DB"   // DB94
VERSION : 0.1
// stored: AutoNumber true, InstanceOfName SCLTestingEnc, InstanceOfType FB
"SCLTestingEnc"
BEGIN
END_DATA_BLOCK

DATA_BLOCK "Blinker_BlowOff"   // DB74
VERSION : 0.1
// stored: AutoNumber true, InstanceOfName Blinker, InstanceOfType FB
"Blinker"
BEGIN
END_DATA_BLOCK

DATA_BLOCK "Blinker_BlueBlinking"   // DB63
VERSION : 0.1
// stored: AutoNumber true, InstanceOfName Blinker, InstanceOfType FB
"Blinker"
BEGIN
END_DATA_BLOCK

DATA_BLOCK "Blinker_BlueConstant"   // DB65
VERSION : 0.1
// stored: AutoNumber true, InstanceOfName Blinker, InstanceOfType FB
"Blinker"
BEGIN
END_DATA_BLOCK

DATA_BLOCK "Blinker_GreenConstant"   // DB81
VERSION : 0.1
// stored: AutoNumber true, InstanceOfName Blinker, InstanceOfType FB
"Blinker"
BEGIN
END_DATA_BLOCK

DATA_BLOCK "BlowOff_Timer_Cleaning"   // DB73
VERSION : 0.1
// stored: AutoNumber true, InstanceOfName BlowOff_Timer, InstanceOfType FB
"BlowOff_Timer"
BEGIN
END_DATA_BLOCK

DATA_BLOCK "BlowOff_Timer_Manual2DB"   // DB86
VERSION : 0.1
// stored: AutoNumber true, InstanceOfName BlowOff_Timer, InstanceOfType FB
"BlowOff_Timer"
BEGIN
END_DATA_BLOCK

DATA_BLOCK "BlowOff_Timer_ManualDB"   // DB83
VERSION : 0.1
// stored: AutoNumber true, InstanceOfName BlowOff_Timer, InstanceOfType FB
"BlowOff_Timer"
BEGIN
END_DATA_BLOCK

DATA_BLOCK "BlowOff_Timer_Prog1"   // DB75
VERSION : 0.1
// stored: AutoNumber true, InstanceOfName BlowOff_Timer, InstanceOfType FB
"BlowOff_Timer"
BEGIN
END_DATA_BLOCK

DATA_BLOCK "FB_EncoderFeedback_Aanvoerband"   // DB78
VERSION : 0.1
// stored: AutoNumber true, InstanceOfName FB_EncoderFeedback_Degree, InstanceOfType FB
"FB_EncoderFeedback_Degree"
BEGIN
END_DATA_BLOCK

DATA_BLOCK "FB_ProductTrigger_1"   // DB67
VERSION : 0.1
// stored: AutoNumber true, InstanceOfName FB_ProductTrigger, InstanceOfType FB
"FB_ProductTrigger"
BEGIN
END_DATA_BLOCK

DATA_BLOCK "FB_SystemTimeCounter_DB_1"   // DB23
VERSION : 0.1
// stored: AutoNumber true, InstanceOfName FB_SystemTimeCounter, InstanceOfType FB
"FB_SystemTimeCounter"
BEGIN
END_DATA_BLOCK

DATA_BLOCK "MC_Move_1"   // DB76
VERSION : 0.1
// stored: AutoNumber true, InstanceOfName MC_Move, InstanceOfType FB
"MC_Move"
BEGIN
END_DATA_BLOCK

DATA_BLOCK "MC_Move_2"   // DB77
VERSION : 0.1
// stored: AutoNumber true, InstanceOfName MC_Move, InstanceOfType FB
"MC_Move"
BEGIN
END_DATA_BLOCK

DATA_BLOCK "MC_Move_DB"   // DB62
VERSION : 0.1
// stored: AutoNumber true, InstanceOfName MC_Move, InstanceOfType FB
"MC_Move"
BEGIN
END_DATA_BLOCK

DATA_BLOCK "MC_Move_Prog.1_1"   // DB59
VERSION : 0.1
// stored: AutoNumber true, InstanceOfName MC_Move, InstanceOfType FB
"MC_Move"
BEGIN
END_DATA_BLOCK

DATA_BLOCK "ProductBuffer_BehindWals"   // DB79
VERSION : 0.1
// stored: AutoNumber true, InstanceOfName ProductBuffer, InstanceOfType FB
"ProductBuffer"
BEGIN
END_DATA_BLOCK

DATA_BLOCK "ProductBuffer_DB"   // DB58
VERSION : 0.1
// stored: AutoNumber true, InstanceOfName ProductBuffer, InstanceOfType FB
"ProductBuffer"
BEGIN
END_DATA_BLOCK

DATA_BLOCK "ProductBuffer_DB_Manual"   // DB85
VERSION : 0.1
// stored: AutoNumber true, InstanceOfName ProductBuffer, InstanceOfType FB
"ProductBuffer"
BEGIN
END_DATA_BLOCK

DATA_BLOCK "ProductBuffer_V2_DB"   // DB66
VERSION : 0.1
// stored: AutoNumber true, InstanceOfName ProductBuffer_V2, InstanceOfType FB
"ProductBuffer_V2"
BEGIN
END_DATA_BLOCK

DATA_BLOCK "ProductBuffer_V2_DB_BehindWals"   // DB82
VERSION : 0.1
// stored: AutoNumber true, InstanceOfName ProductBuffer_V2, InstanceOfType FB
"ProductBuffer_V2"
BEGIN
END_DATA_BLOCK

DATA_BLOCK "Programma 1 - Test_DB"   // DB64
VERSION : 0.1
// stored: AutoNumber true, InstanceOfName Programma 1 - Test, InstanceOfType FB
"Programma 1 - Test"
BEGIN
END_DATA_BLOCK

DATA_BLOCK "ResetOuputs_Function_Rest"   // DB29
VERSION : 0.1
// stored: AutoNumber true, InstanceOfName ResetOuputs_Function, InstanceOfType FB
"ResetOuputs_Function"
BEGIN
END_DATA_BLOCK

DATA_BLOCK "FB_SystemTimeCounter_DB"   // DB69
VERSION : 0.1
// stored: AutoNumber true, InstanceOfName FB_SystemTimeCounter, InstanceOfType FB
"FB_SystemTimeCounter"
BEGIN
END_DATA_BLOCK

DATA_BLOCK "Blinker_Start"   // DB71
VERSION : 0.1
// stored: AutoNumber true, InstanceOfName Blinker, InstanceOfType FB
"Blinker"
BEGIN
END_DATA_BLOCK

DATA_BLOCK "SwitchBlockAxisPosition_DB"   // DB39
VERSION : 0.1
// stored: AutoNumber true, InstanceOfName SwitchBlockAxisPosition, InstanceOfType FB
"SwitchBlockAxisPosition"
BEGIN
END_DATA_BLOCK

DATA_BLOCK "2in-1out_Block_LED-Estop"   // DB1
VERSION : 0.1
// stored: AutoNumber true, InstanceOfName 2in-1out_Block, InstanceOfType FB
"2in-1out_Block"
BEGIN
END_DATA_BLOCK

DATA_BLOCK "Alarm_Axis_Position_Function_Infeed"   // DB43
VERSION : 0.1
// stored: AutoNumber true, InstanceOfName Alarm_Axis_Position_Function, InstanceOfType FB
"Alarm_Axis_Position_Function"
BEGIN
END_DATA_BLOCK

DATA_BLOCK "Alarm_Axis_Position_Function_Wals"   // DB41
VERSION : 0.1
// stored: AutoNumber true, InstanceOfName Alarm_Axis_Position_Function, InstanceOfType FB
"Alarm_Axis_Position_Function"
BEGIN
END_DATA_BLOCK

DATA_BLOCK "Alarm_Axis_Position_Function_Wals1"   // DB42
VERSION : 0.1
// stored: AutoNumber true, InstanceOfName Alarm_Axis_Position_Function, InstanceOfType FB
"Alarm_Axis_Position_Function"
BEGIN
END_DATA_BLOCK

DATA_BLOCK "Delayed_Message_Function_Magazine"   // DB38
VERSION : 0.1
// stored: AutoNumber true, InstanceOfName Delayed_Message_Function, InstanceOfType FB
"Delayed_Message_Function"
BEGIN
END_DATA_BLOCK

DATA_BLOCK "DriveConfirmation_Function_Axis 3"   // DB47
VERSION : 0.1
// stored: AutoNumber true, InstanceOfName DriveConfirmation_Function, InstanceOfType FB
"DriveConfirmation_Function"
BEGIN
END_DATA_BLOCK

DATA_BLOCK "DriveConfirmation_Function_Axis 4"   // DB48
VERSION : 0.1
// stored: AutoNumber true, InstanceOfName DriveConfirmation_Function, InstanceOfType FB
"DriveConfirmation_Function"
BEGIN
END_DATA_BLOCK

DATA_BLOCK "DriveConfirmation_Function_Axis 5"   // DB49
VERSION : 0.1
// stored: AutoNumber true, InstanceOfName DriveConfirmation_Function, InstanceOfType FB
"DriveConfirmation_Function"
BEGIN
END_DATA_BLOCK

DATA_BLOCK "DriveConfirmation_Function_Axis1"   // DB45
VERSION : 0.1
// stored: AutoNumber true, InstanceOfName DriveConfirmation_Function, InstanceOfType FB
"DriveConfirmation_Function"
BEGIN
END_DATA_BLOCK

DATA_BLOCK "DriveConfirmation_Function_Axis2"   // DB46
VERSION : 0.1
// stored: AutoNumber true, InstanceOfName DriveConfirmation_Function, InstanceOfType FB
"DriveConfirmation_Function"
BEGIN
END_DATA_BLOCK

DATA_BLOCK "ESB_Buzzer_Block"   // DB33
VERSION : 0.1
// stored: AutoNumber true, InstanceOfName ESB_Flash_Warning_Block, InstanceOfType FB
"ESB_Flash_Warning_Block"
BEGIN
END_DATA_BLOCK

DATA_BLOCK "ESB_Lamp_Block"   // DB34
VERSION : 0.1
// stored: AutoNumber true, InstanceOfName ESB_Flash_Warning_Block, InstanceOfType FB
"ESB_Flash_Warning_Block"
BEGIN
END_DATA_BLOCK

DATA_BLOCK "Ouput_Function_1_Drive1"   // DB4
VERSION : 0.1
// stored: AutoNumber true, InstanceOfName Ouput_Function_1, InstanceOfType FB
"Ouput_Function_1"
BEGIN
END_DATA_BLOCK

DATA_BLOCK "Ouput_Function_1_Drive2"   // DB8
VERSION : 0.1
// stored: AutoNumber true, InstanceOfName Ouput_Function_1, InstanceOfType FB
"Ouput_Function_1"
BEGIN
END_DATA_BLOCK

DATA_BLOCK "Ouput_Function_1_Drive3"   // DB12
VERSION : 0.1
// stored: AutoNumber true, InstanceOfName Ouput_Function_1, InstanceOfType FB
"Ouput_Function_1"
BEGIN
END_DATA_BLOCK

DATA_BLOCK "Ouput_Function_1_Drive4"   // DB17
VERSION : 0.1
// stored: AutoNumber true, InstanceOfName Ouput_Function_1, InstanceOfType FB
"Ouput_Function_1"
BEGIN
END_DATA_BLOCK

DATA_BLOCK "Ouput_Function_1_Drive5"   // DB18
VERSION : 0.1
// stored: AutoNumber true, InstanceOfName Ouput_Function_1, InstanceOfType FB
"Ouput_Function_1"
BEGIN
END_DATA_BLOCK

DATA_BLOCK "Ouput_Function_1_Valve1"   // DB19
VERSION : 0.1
// stored: AutoNumber true, InstanceOfName Ouput_Function_1, InstanceOfType FB
"Ouput_Function_1"
BEGIN
END_DATA_BLOCK

DATA_BLOCK "Ouput_Function_1_Valve2"   // DB25
VERSION : 0.1
// stored: AutoNumber true, InstanceOfName Ouput_Function_1, InstanceOfType FB
"Ouput_Function_1"
BEGIN
END_DATA_BLOCK

DATA_BLOCK "Ouput_Function_1_Valve3"   // DB26
VERSION : 0.1
// stored: AutoNumber true, InstanceOfName Ouput_Function_1, InstanceOfType FB
"Ouput_Function_1"
BEGIN
END_DATA_BLOCK

DATA_BLOCK "Ouput_Function_1_Valve4"   // DB27
VERSION : 0.1
// stored: AutoNumber true, InstanceOfName Ouput_Function_1, InstanceOfType FB
"Ouput_Function_1"
BEGIN
END_DATA_BLOCK

DATA_BLOCK "Ouput_Function_1_Valve5"   // DB28
VERSION : 0.1
// stored: AutoNumber true, InstanceOfName Ouput_Function_1, InstanceOfType FB
"Ouput_Function_1"
BEGIN
END_DATA_BLOCK

DATA_BLOCK "Override_Block_Safety_1"   // DB3
VERSION : 0.1
// stored: AutoNumber true, InstanceOfName Override_Block_Safety, InstanceOfType FB
"Override_Block_Safety"
BEGIN
END_DATA_BLOCK

DATA_BLOCK "EncoderFeedback_Band"   // DB89
VERSION : 0.1
// stored: AutoNumber true, InstanceOfName FB_EncoderFeedback_Lineair, InstanceOfType FB
"FB_EncoderFeedback_Lineair"
BEGIN
END_DATA_BLOCK

DATA_BLOCK "FB_Encoder64Bit_DB"   // DB92
VERSION : 0.1
// stored: AutoNumber true, InstanceOfName FB_Encoder64Bit, InstanceOfType FB
"FB_Encoder64Bit"
BEGIN
END_DATA_BLOCK

DATA_BLOCK "MC_Jog_OB1"   // DB56
VERSION : 0.1
// stored: AutoNumber true, InstanceOfName MC_Jog, InstanceOfType FB
"MC_Jog"
BEGIN
END_DATA_BLOCK

DATA_BLOCK "MC_Move_Prog.1"   // DB54
VERSION : 0.1
// stored: AutoNumber true, InstanceOfName MC_Move, InstanceOfType FB
"MC_Move"
BEGIN
END_DATA_BLOCK

DATA_BLOCK "BlowOffStartTimer"   // DB98
// stored: AutoNumber true, InstanceOfName TOF_SFB, OfSystemLibElement TOF, OfSystemLibVersion 1.0
"TOF_SFB"
   // VAR_INPUT
   //    IN : Bool;
   //    PT : Time;
   // END_VAR
   // VAR_OUTPUT
   //    Q : Bool;
   //    ET : Time;
   // END_VAR
   // VAR RETAIN
   //    STATE : Byte;
   //    STIME : Time;
   //    ATIME : Time;
   // END_VAR
BEGIN
END_DATA_BLOCK

DATA_BLOCK "BrakeTimer"   // DB53
// stored: AutoNumber true, InstanceOfName TON_SFB, OfSystemLibElement TON, OfSystemLibVersion 1.0
"TON_SFB"
   // VAR_INPUT
   //    IN : Bool;
   //    PT : Time;
   // END_VAR
   // VAR_OUTPUT
   //    Q : Bool;
   //    ET : Time;
   // END_VAR
   // VAR RETAIN
   //    STATE : Byte;
   //    STIME : Time;
   //    ATIME : Time;
   // END_VAR
BEGIN
END_DATA_BLOCK

DATA_BLOCK "BrakeTimerManual"   // DB55
// stored: AutoNumber true, InstanceOfName TOF_SFB, OfSystemLibElement TOF, OfSystemLibVersion 1.0
"TOF_SFB"
   // VAR_INPUT
   //    IN : Bool;
   //    PT : Time;
   // END_VAR
   // VAR_OUTPUT
   //    Q : Bool;
   //    ET : Time;
   // END_VAR
   // VAR RETAIN
   //    STATE : Byte;
   //    STIME : Time;
   //    ATIME : Time;
   // END_VAR
BEGIN
END_DATA_BLOCK

DATA_BLOCK "ConfirimationDrivesTimer"   // DB44
// stored: AutoNumber true, InstanceOfName TON_SFB, OfSystemLibElement TON, OfSystemLibVersion 1.0
"TON_SFB"
   // VAR_INPUT
   //    IN : Bool;
   //    PT : Time;
   // END_VAR
   // VAR_OUTPUT
   //    Q : Bool;
   //    ET : Time;
   // END_VAR
   // VAR RETAIN
   //    STATE : Byte;
   //    STIME : Time;
   //    ATIME : Time;
   // END_VAR
BEGIN
END_DATA_BLOCK

DATA_BLOCK "Delayed_Message_Function_Timer"   // DB35
// stored: AutoNumber true, InstanceOfName TON_SFB, OfSystemLibElement TON, OfSystemLibVersion 1.0
"TON_SFB"
   // VAR_INPUT
   //    IN : Bool;
   //    PT : Time;
   // END_VAR
   // VAR_OUTPUT
   //    Q : Bool;
   //    ET : Time;
   // END_VAR
   // VAR RETAIN
   //    STATE : Byte;
   //    STIME : Time;
   //    ATIME : Time;
   // END_VAR
BEGIN
END_DATA_BLOCK

DATA_BLOCK "IEC_Timer_0_DB"   // DB31
// stored: AutoNumber true, InstanceOfName TON_SFB, OfSystemLibElement TON, OfSystemLibVersion 1.0
"TON_SFB"
   // VAR_INPUT
   //    IN : Bool;
   //    PT : Time;
   // END_VAR
   // VAR_OUTPUT
   //    Q : Bool;
   //    ET : Time;
   // END_VAR
   // VAR RETAIN
   //    STATE : Byte;
   //    STIME : Time;
   //    ATIME : Time;
   // END_VAR
BEGIN
END_DATA_BLOCK

DATA_BLOCK "IEC_Timer_0_DB_1"   // DB60
// stored: AutoNumber true, InstanceOfName TOF_SFB, OfSystemLibElement TOF, OfSystemLibVersion 1.0
"TOF_SFB"
   // VAR_INPUT
   //    IN : Bool;
   //    PT : Time;
   // END_VAR
   // VAR_OUTPUT
   //    Q : Bool;
   //    ET : Time;
   // END_VAR
   // VAR RETAIN
   //    STATE : Byte;
   //    STIME : Time;
   //    ATIME : Time;
   // END_VAR
BEGIN
END_DATA_BLOCK

DATA_BLOCK "IEC_Timer_0_DB_2"   // DB9
// stored: AutoNumber true, InstanceOfName TOF_SFB, OfSystemLibElement TOF, OfSystemLibVersion 1.0
"TOF_SFB"
   // VAR_INPUT
   //    IN : Bool;
   //    PT : Time;
   // END_VAR
   // VAR_OUTPUT
   //    Q : Bool;
   //    ET : Time;
   // END_VAR
   // VAR RETAIN
   //    STATE : Byte;
   //    STIME : Time;
   //    ATIME : Time;
   // END_VAR
BEGIN
END_DATA_BLOCK

DATA_BLOCK "IEC_Timer_0_DB_3"   // DB91
// stored: AutoNumber true, InstanceOfName TON_SFB, OfSystemLibElement TON, OfSystemLibVersion 1.0
"TON_SFB"
   // VAR_INPUT
   //    IN : Bool;
   //    PT : Time;
   // END_VAR
   // VAR_OUTPUT
   //    Q : Bool;
   //    ET : Time;
   // END_VAR
   // VAR RETAIN
   //    STATE : Byte;
   //    STIME : Time;
   //    ATIME : Time;
   // END_VAR
BEGIN
END_DATA_BLOCK

DATA_BLOCK "Move2Done"   // DB88
// stored: AutoNumber true, InstanceOfName TON_SFB, OfSystemLibElement TON, OfSystemLibVersion 1.0
"TON_SFB"
   // VAR_INPUT
   //    IN : Bool;
   //    PT : Time;
   // END_VAR
   // VAR_OUTPUT
   //    Q : Bool;
   //    ET : Time;
   // END_VAR
   // VAR RETAIN
   //    STATE : Byte;
   //    STIME : Time;
   //    ATIME : Time;
   // END_VAR
BEGIN
END_DATA_BLOCK

DATA_BLOCK "NotEnoughProducts"   // DB84
// stored: AutoNumber true, InstanceOfName TON_SFB, OfSystemLibElement TON, OfSystemLibVersion 1.0
"TON_SFB"
   // VAR_INPUT
   //    IN : Bool;
   //    PT : Time;
   // END_VAR
   // VAR_OUTPUT
   //    Q : Bool;
   //    ET : Time;
   // END_VAR
   // VAR RETAIN
   //    STATE : Byte;
   //    STIME : Time;
   //    ATIME : Time;
   // END_VAR
BEGIN
END_DATA_BLOCK

DATA_BLOCK "ProductBufferTimer"   // DB80
// stored: AutoNumber true, InstanceOfName TON_SFB, OfSystemLibElement TON, OfSystemLibVersion 1.0
"TON_SFB"
   // VAR_INPUT
   //    IN : Bool;
   //    PT : Time;
   // END_VAR
   // VAR_OUTPUT
   //    Q : Bool;
   //    ET : Time;
   // END_VAR
   // VAR RETAIN
   //    STATE : Byte;
   //    STIME : Time;
   //    ATIME : Time;
   // END_VAR
BEGIN
END_DATA_BLOCK

DATA_BLOCK "ProductCounter"   // DB21
// stored: AutoNumber true, InstanceOfName CTU_SFB, OfSystemLibElement CTU, OfSystemLibVersion 1.0
"CTU_SFB"
   // VAR_INPUT
   //    CU : Bool;
   //    R : Bool;
   //    PV : Int;
   // END_VAR
   // VAR_OUTPUT
   //    Q : Bool;
   //    CV : Int;
   // END_VAR
   // VAR RETAIN
   //    CUO : Bool;
   // END_VAR
BEGIN
END_DATA_BLOCK

DATA_BLOCK "RestAferReferenceRun"   // DB52
// stored: AutoNumber true, InstanceOfName TON_SFB, OfSystemLibElement TON, OfSystemLibVersion 1.0
"TON_SFB"
   // VAR_INPUT
   //    IN : Bool;
   //    PT : Time;
   // END_VAR
   // VAR_OUTPUT
   //    Q : Bool;
   //    ET : Time;
   // END_VAR
   // VAR RETAIN
   //    STATE : Byte;
   //    STIME : Time;
   //    ATIME : Time;
   // END_VAR
BEGIN
END_DATA_BLOCK

DATA_BLOCK "SafetyTimer"   // DB16
// stored: AutoNumber true, InstanceOfName TON_SFB, OfSystemLibElement TON, OfSystemLibVersion 1.0
"TON_SFB"
   // VAR_INPUT
   //    IN : Bool;
   //    PT : Time;
   // END_VAR
   // VAR_OUTPUT
   //    Q : Bool;
   //    ET : Time;
   // END_VAR
   // VAR RETAIN
   //    STATE : Byte;
   //    STIME : Time;
   //    ATIME : Time;
   // END_VAR
BEGIN
END_DATA_BLOCK

DATA_BLOCK "StartDelayTimer"   // DB57
// stored: AutoNumber true, InstanceOfName TON_SFB, OfSystemLibElement TON, OfSystemLibVersion 1.0
"TON_SFB"
   // VAR_INPUT
   //    IN : Bool;
   //    PT : Time;
   // END_VAR
   // VAR_OUTPUT
   //    Q : Bool;
   //    ET : Time;
   // END_VAR
   // VAR RETAIN
   //    STATE : Byte;
   //    STIME : Time;
   //    ATIME : Time;
   // END_VAR
BEGIN
END_DATA_BLOCK

DATA_BLOCK "TimerOffDelayMove2"   // DB97
// stored: AutoNumber true, InstanceOfName TOF_SFB, OfSystemLibElement TOF, OfSystemLibVersion 1.0
"TOF_SFB"
   // VAR_INPUT
   //    IN : Bool;
   //    PT : Time;
   // END_VAR
   // VAR_OUTPUT
   //    Q : Bool;
   //    ET : Time;
   // END_VAR
   // VAR RETAIN
   //    STATE : Byte;
   //    STIME : Time;
   //    ATIME : Time;
   // END_VAR
BEGIN
END_DATA_BLOCK

DATA_BLOCK "Timer_0_5s"   // DB30
// stored: AutoNumber true, InstanceOfName TON_SFB, OfSystemLibElement TON, OfSystemLibVersion 1.0
"TON_SFB"
   // VAR_INPUT
   //    IN : Bool;
   //    PT : Time;
   // END_VAR
   // VAR_OUTPUT
   //    Q : Bool;
   //    ET : Time;
   // END_VAR
   // VAR RETAIN
   //    STATE : Byte;
   //    STIME : Time;
   //    ATIME : Time;
   // END_VAR
BEGIN
END_DATA_BLOCK

DATA_BLOCK "Timer_Aanvoerband"   // DB7
// stored: AutoNumber true, InstanceOfName TON_SFB, OfSystemLibElement TON, OfSystemLibVersion 1.0
"TON_SFB"
   // VAR_INPUT
   //    IN : Bool;
   //    PT : Time;
   // END_VAR
   // VAR_OUTPUT
   //    Q : Bool;
   //    ET : Time;
   // END_VAR
   // VAR RETAIN
   //    STATE : Byte;
   //    STIME : Time;
   //    ATIME : Time;
   // END_VAR
BEGIN
END_DATA_BLOCK

DATA_BLOCK "Timer_AxisCheck"   // DB40
// stored: AutoNumber true, InstanceOfName TON_SFB, OfSystemLibElement TON, OfSystemLibVersion 1.0
"TON_SFB"
   // VAR_INPUT
   //    IN : Bool;
   //    PT : Time;
   // END_VAR
   // VAR_OUTPUT
   //    Q : Bool;
   //    ET : Time;
   // END_VAR
   // VAR RETAIN
   //    STATE : Byte;
   //    STIME : Time;
   //    ATIME : Time;
   // END_VAR
BEGIN
END_DATA_BLOCK

DATA_BLOCK "Timer_ProductInterval"   // DB20
// stored: AutoNumber true, InstanceOfName TON_SFB, OfSystemLibElement TON, OfSystemLibVersion 1.0
"TON_SFB"
   // VAR_INPUT
   //    IN : Bool;
   //    PT : Time;
   // END_VAR
   // VAR_OUTPUT
   //    Q : Bool;
   //    ET : Time;
   // END_VAR
   // VAR RETAIN
   //    STATE : Byte;
   //    STIME : Time;
   //    ATIME : Time;
   // END_VAR
BEGIN
END_DATA_BLOCK

DATA_BLOCK "Timer_Retourband"   // DB70
// stored: AutoNumber true, InstanceOfName TON_SFB, OfSystemLibElement TON, OfSystemLibVersion 1.0
"TON_SFB"
   // VAR_INPUT
   //    IN : Bool;
   //    PT : Time;
   // END_VAR
   // VAR_OUTPUT
   //    Q : Bool;
   //    ET : Time;
   // END_VAR
   // VAR RETAIN
   //    STATE : Byte;
   //    STIME : Time;
   //    ATIME : Time;
   // END_VAR
BEGIN
END_DATA_BLOCK

DATA_BLOCK "Timer_Retourband_Off"   // DB72
// stored: AutoNumber true, InstanceOfName TOF_SFB, OfSystemLibElement TOF, OfSystemLibVersion 1.0
"TOF_SFB"
   // VAR_INPUT
   //    IN : Bool;
   //    PT : Time;
   // END_VAR
   // VAR_OUTPUT
   //    Q : Bool;
   //    ET : Time;
   // END_VAR
   // VAR RETAIN
   //    STATE : Byte;
   //    STIME : Time;
   //    ATIME : Time;
   // END_VAR
BEGIN
END_DATA_BLOCK

DATA_BLOCK "Timer_Signal_1"   // DB36
// stored: AutoNumber true, InstanceOfName TP_SFB, OfSystemLibElement TP, OfSystemLibVersion 1.0
"TP_SFB"
   // VAR_INPUT
   //    IN : Bool;
   //    PT : Time;
   // END_VAR
   // VAR_OUTPUT
   //    Q : Bool;
   //    ET : Time;
   // END_VAR
   // VAR RETAIN
   //    STATE : Byte;
   //    STIME : Time;
   //    ATIME : Time;
   // END_VAR
BEGIN
END_DATA_BLOCK

DATA_BLOCK "Timer_Signal_2"   // DB37
// stored: AutoNumber true, InstanceOfName TON_SFB, OfSystemLibElement TON, OfSystemLibVersion 1.0
"TON_SFB"
   // VAR_INPUT
   //    IN : Bool;
   //    PT : Time;
   // END_VAR
   // VAR_OUTPUT
   //    Q : Bool;
   //    ET : Time;
   // END_VAR
   // VAR RETAIN
   //    STATE : Byte;
   //    STIME : Time;
   //    ATIME : Time;
   // END_VAR
BEGIN
END_DATA_BLOCK

DATA_BLOCK "Timer_Trilgoten"   // DB5
// stored: AutoNumber true, InstanceOfName TON_SFB, OfSystemLibElement TON, OfSystemLibVersion 1.0
"TON_SFB"
   // VAR_INPUT
   //    IN : Bool;
   //    PT : Time;
   // END_VAR
   // VAR_OUTPUT
   //    Q : Bool;
   //    ET : Time;
   // END_VAR
   // VAR RETAIN
   //    STATE : Byte;
   //    STIME : Time;
   //    ATIME : Time;
   // END_VAR
BEGIN
END_DATA_BLOCK

DATA_BLOCK "TotalProductsCounter"   // DB22
// stored: AutoNumber true, InstanceOfName CTU_SFB, OfSystemLibElement CTU, OfSystemLibVersion 1.0
"CTU_SFB"
   // VAR_INPUT
   //    CU : Bool;
   //    R : Bool;
   //    PV : Int;
   // END_VAR
   // VAR_OUTPUT
   //    Q : Bool;
   //    CV : Int;
   // END_VAR
   // VAR RETAIN
   //    CUO : Bool;
   // END_VAR
BEGIN
END_DATA_BLOCK

DATA_BLOCK "Uitlooptimer_Aanvoerband"   // DB10
// stored: AutoNumber true, InstanceOfName TON_SFB, OfSystemLibElement TON, OfSystemLibVersion 1.0
"TON_SFB"
   // VAR_INPUT
   //    IN : Bool;
   //    PT : Time;
   // END_VAR
   // VAR_OUTPUT
   //    Q : Bool;
   //    ET : Time;
   // END_VAR
   // VAR RETAIN
   //    STATE : Byte;
   //    STIME : Time;
   //    ATIME : Time;
   // END_VAR
BEGIN
END_DATA_BLOCK

DATA_BLOCK "Uitlooptimer_Trilgoten"   // DB11
// stored: AutoNumber true, InstanceOfName TON_SFB, OfSystemLibElement TON, OfSystemLibVersion 1.0
"TON_SFB"
   // VAR_INPUT
   //    IN : Bool;
   //    PT : Time;
   // END_VAR
   // VAR_OUTPUT
   //    Q : Bool;
   //    ET : Time;
   // END_VAR
   // VAR RETAIN
   //    STATE : Byte;
   //    STIME : Time;
   //    ATIME : Time;
   // END_VAR
BEGIN
END_DATA_BLOCK

DATA_BLOCK "WarningTimer2"   // DB32
// stored: AutoNumber true, InstanceOfName TON_SFB, OfSystemLibElement TON, OfSystemLibVersion 1.0
"TON_SFB"
   // VAR_INPUT
   //    IN : Bool;
   //    PT : Time;
   // END_VAR
   // VAR_OUTPUT
   //    Q : Bool;
   //    ET : Time;
   // END_VAR
   // VAR RETAIN
   //    STATE : Byte;
   //    STIME : Time;
   //    ATIME : Time;
   // END_VAR
BEGIN
END_DATA_BLOCK

DATA_BLOCK "WarningTimer3"   // DB61
// stored: AutoNumber true, InstanceOfName TON_SFB, OfSystemLibElement TON, OfSystemLibVersion 1.0
"TON_SFB"
   // VAR_INPUT
   //    IN : Bool;
   //    PT : Time;
   // END_VAR
   // VAR_OUTPUT
   //    Q : Bool;
   //    ET : Time;
   // END_VAR
   // VAR RETAIN
   //    STATE : Byte;
   //    STIME : Time;
   //    ATIME : Time;
   // END_VAR
BEGIN
END_DATA_BLOCK

DATA_BLOCK "Blinker_SimulateSensor_DB"   // DB100
VERSION : 0.1
// stored: AutoNumber true, InstanceOfName Blinker, InstanceOfType FB
"Blinker"
BEGIN
END_DATA_BLOCK

DATA_BLOCK "Blinker_Yellow"   // DB102
VERSION : 0.1
// stored: AutoNumber true, InstanceOfName Blinker, InstanceOfType FB
"Blinker"
BEGIN
END_DATA_BLOCK

DATA_BLOCK "BlowOffTimerV2"   // DB13
// stored: AutoNumber true, InstanceOfName TOF_SFB, OfSystemLibElement TOF, OfSystemLibVersion 1.0
"TOF_SFB"
   // VAR_INPUT
   //    IN : Bool;
   //    PT : Time;
   // END_VAR
   // VAR_OUTPUT
   //    Q : Bool;
   //    ET : Time;
   // END_VAR
   // VAR RETAIN
   //    STATE : Byte;
   //    STIME : Time;
   //    ATIME : Time;
   // END_VAR
BEGIN
END_DATA_BLOCK

DATA_BLOCK "EncoderET200S1COUNT_DB"   // DB87
// stored: AutoNumber true, InstanceOfName EncoderET200S1COUNT, OfSystemLibElement EncoderET200S1COUNT, OfSystemLibVersion 2.3
"EncoderET200S1COUNT"
   // VAR_INPUT
   //    EncErr : Bool;
   //    DOut_1 : Bool;
   //    DOut_2 : Bool;
   // END_VAR
   // VAR_OUTPUT
   //    DIn : Bool;
   // END_VAR
   // VAR_IN_OUT
   //    Axis : Struct
   //       Sample_T : Real;
   //       AxisType : Bool;
   //       EncoderType : Bool;
   //       Sim : Bool;
   //       AxisLimitMax : Real;
   //       AxisLimitMin : Real;
   //       MaxVelocity : Real;
   //       MaxAcceleration : Real;
   //       MaxDeceleration : Real;
   //       MonTimeTargetAppr : Real;
   //       TargetRange : Real;
   //       StandstillRange : Real;
   //       MaxFollowingDist : Real;
   //       MonitorTargetAppr : Bool;
   //       SWLimitEnable : Bool;
   //       FactorP : Real;
   //       ManVelocity : Real;
   //       ManEnable : Bool;
   //       EmergencyDec : Real;
   //       InputModuleInAddr : Int;
   //       InputModuleOutAddr : Int;
   //       InputChannelNo : Int;
   //       StepsPerRev : DInt;
   //       DisplacementPerRev : Real;
   //       NumberRevs : Int;
   //       PolarityEncoder : Int;
   //       PositionOffset : DInt;
   //       OutputModuleOutAddr : Int;
   //       OutputModuleInAddr : Int;
   //       OutputChannelNo : Int;
   //       PolarityDrive : Int;
   //       DriveInputAtMaxVel : Real;
   //       OffsetCompensation : Real;
   //       DriveInputAt100 : Real;
   //       Override : Real;
   //       ActPosition : Real;
   //       FollowingDistance : Real;
   //       RemainingDistance : Real;
   //       NomVelocity : Real;
   //       ActVelocity : Real;
   //       Sync : Bool;
   //       Error : Bool;
   //       ErrorAck : Bool;
   //       AxisState : Int;
   //       Err : Struct
   //          SWLimitMinExceeded : Bool;
   //          SWLimitMaxExceeded : Bool;
   //          TargetErr : Bool;
   //          NoSync : Bool;
   //          DirectionErr : Bool;
   //          DataErr : Bool;
   //          StartErr : Bool;
   //          DistanceErr : Bool;
   //          MasterErr : Bool;
   //          bit09 : Bool;
   //          bit10 : Bool;
   //          bit11 : Bool;
   //          bit12 : Bool;
   //          bit13 : Bool;
   //          bit14 : Bool;
   //          bit15 : Bool;
   //          StoppedMotion : Bool;
   //          EnableDriveErr : Bool;
   //          FollowingDistErr : Bool;
   //          StandstillErr : Bool;
   //          TargetApproachErr : Bool;
   //          EncoderErr : Bool;
   //          OutputErr : Bool;
   //          ConfigErr : Bool;
   //          DriveErr : Bool;
   //          bit25 : Bool;
   //          bit26 : Bool;
   //          bit27 : Bool;
   //          bit28 : Bool;
   //          bit29 : Bool;
   //          bit30 : Bool;
   //          bit31 : Bool;
   //       END_STRUCT;
   //       Config : Struct
   //          Err_AxisLimit : Bool;
   //          Err_MaxVelocity : Bool;
   //          Err_MaxAcceleration : Bool;
   //          Err_MaxDeceleration : Bool;
   //          Err_MonTimeTargetAppr : Bool;
   //          Err_TargetRange : Bool;
   //          Err_StandstillRange : Bool;
   //          Err_MaxFollowingDist : Bool;
   //          Err_EmergencyDec : Bool;
   //          Err_StepsPerRev : Bool;
   //          Err_DisplacementPerRev : Bool;
   //          Err_NumberRevs : Bool;
   //          Err_PolarityEncoder : Bool;
   //          Err_PolarityDrive : Bool;
   //          Err_DriveInputAtMaxVel : Bool;
   //          Err_AxisLength : Bool;
   //          Err_EncoderRange : Bool;
   //          Err_MaxVelRotaryAxis : Bool;
   //          Err_DriveInputAt100 : Bool;
   //       END_STRUCT;
   //       EncoderValue : DInt;
   //       RefPoint : Real;
   //       OutVelocity : Real;
   //       LastNomPosition : Real;
   //       LastNomVelocity : Real;
   //       LastNomDeceleration : Real;
   //       InternalNomPosition : Real;
   //       InternalActPos : Real;
   //       InternalPosOffset : Real;
   //       aufl : Real;
   //       AchsLaenge : Real;
   //       AchsLaenge_DI : DInt;
   //       AbsGeberLaenge_DI : DInt;
   //       LageIstwert_DI : DInt;
   //       Coord : DInt;
   //       DoneRef : Bool;
   //       EinInitLaeuft : Bool;
   //       AusInitLaeuft : Bool;
   //       EinQuittungLaeuft : Bool;
   //       AusQuittungLaeuft : Bool;
   //       EintreiberFahrbereit : Bool;
   //       ExecRef : Int;
   //       VLastNomPosition : Real;
   //       VLastNomVelocity : Real;
   //       LastInternalPosOffset : Real;
   //       RundKorrektur : Real;
   //       LastRundKorrektur : Real;
   //       LengthUnit : String[4];
   //       InputModuleType : String[24];
   //       OutputModuleType : String[24];
   //       Init : Struct
   //          I0 : Bool;
   //          I1 : Bool;
   //          I2 : Bool;
   //          I3 : Bool;
   //          I4 : Bool;
   //          I5 : Bool;
   //          I6 : Bool;
   //          I7 : Bool;
   //          I8 : Bool;
   //          I9 : Bool;
   //          I10 : Bool;
   //          I11 : Bool;
   //          I12 : Bool;
   //          I13 : Bool;
   //          I14 : Bool;
   //          I15 : Bool;
   //          I16 : Bool;
   //          I17 : Bool;
   //          I18 : Bool;
   //          I19 : Bool;
   //          I20 : Bool;
   //          I21 : Bool;
   //          I22 : Bool;
   //          I23 : Bool;
   //          I24 : Bool;
   //          I25 : Bool;
   //          I26 : Bool;
   //          I27 : Bool;
   //          I28 : Bool;
   //          I29 : Bool;
   //          I30 : Bool;
   //          I31 : Bool;
   //       END_STRUCT;
   //    END_STRUCT;
   //    Init : Bool;
   // END_VAR
   // VAR RETAIN
   //    Status : Struct
   //       STS_LOAD : Bool;
   //       ERR_LOAD : Bool;
   //       RES_STS_A : Bool;
   //       ERR_ENCODER : Bool;
   //       ERR_DO2 : Bool;
   //       ERR_PARA : Bool;
   //       ERR_DO1 : Bool;
   //       ERR_24V : Bool;
   //       STS_GATE : Bool;
   //       STS_DI : Bool;
   //       bit18 : Bool;
   //       STS_DO1 : Bool;
   //       STS_DO2 : Bool;
   //       bit21 : Bool;
   //       STS_C_UP : Bool;
   //       STS_C_DN : Bool;
   //       STS_SYN : Bool;
   //       bit09 : Bool;
   //       bit10 : Bool;
   //       STS_CMP1 : Bool;
   //       STS_CMP2 : Bool;
   //       STS_OFLW : Bool;
   //       STS_UFLW : Bool;
   //       STS_ND : Bool;
   //       byte3 : Byte;
   //    END_STRUCT;
   //    GeberAlt_DI : DInt;
   //    Addr_ActPos_DI : Int;
   //    Addr_Status : Int;
   //    Addr_LoadVal_DI : Int;
   //    Addr_Steuer : Int;
   //    Richtungsanpassung : Int;
   //    v_Faktor : Real;
   //    MaxZahl : DInt;
   //    MaxZahlHalb : DInt;
   //    PASteuer : Word;
   //    RefPointInt : Real;
   //    LoadVal_DW : DWord;
   //    EncoderZustand : Int;
   //    RefZustand : Int;
   //    aufl : Real;
   //    EncErr_alt : Bool;
   //    Taktsynchron : Bool;
   // END_VAR
BEGIN
END_DATA_BLOCK

DATA_BLOCK "MC_Simulation_DB"   // DB99
// stored: AutoNumber true, InstanceOfName MC_Simulation, OfSystemLibElement MC_Simulation, OfSystemLibVersion 2.1
"MC_Simulation"
   // VAR_IN_OUT
   //    Axis : Struct
   //       Sample_T : Real;
   //       AxisType : Bool;
   //       EncoderType : Bool;
   //       Sim : Bool;
   //       AxisLimitMax : Real;
   //       AxisLimitMin : Real;
   //       MaxVelocity : Real;
   //       MaxAcceleration : Real;
   //       MaxDeceleration : Real;
   //       MonTimeTargetAppr : Real;
   //       TargetRange : Real;
   //       StandstillRange : Real;
   //       MaxFollowingDist : Real;
   //       MonitorTargetAppr : Bool;
   //       SWLimitEnable : Bool;
   //       FactorP : Real;
   //       ManVelocity : Real;
   //       ManEnable : Bool;
   //       EmergencyDec : Real;
   //       InputModuleInAddr : Int;
   //       InputModuleOutAddr : Int;
   //       InputChannelNo : Int;
   //       StepsPerRev : DInt;
   //       DisplacementPerRev : Real;
   //       NumberRevs : Int;
   //       PolarityEncoder : Int;
   //       PositionOffset : DInt;
   //       OutputModuleOutAddr : Int;
   //       OutputModuleInAddr : Int;
   //       OutputChannelNo : Int;
   //       PolarityDrive : Int;
   //       DriveInputAtMaxVel : Real;
   //       OffsetCompensation : Real;
   //       DriveInputAt100 : Real;
   //       Override : Real;
   //       ActPosition : Real;
   //       FollowingDistance : Real;
   //       RemainingDistance : Real;
   //       NomVelocity : Real;
   //       ActVelocity : Real;
   //       Sync : Bool;
   //       Error : Bool;
   //       ErrorAck : Bool;
   //       AxisState : Int;
   //       Err : Struct
   //          SWLimitMinExceeded : Bool;
   //          SWLimitMaxExceeded : Bool;
   //          TargetErr : Bool;
   //          NoSync : Bool;
   //          DirectionErr : Bool;
   //          DataErr : Bool;
   //          StartErr : Bool;
   //          DistanceErr : Bool;
   //          MasterErr : Bool;
   //          bit09 : Bool;
   //          bit10 : Bool;
   //          bit11 : Bool;
   //          bit12 : Bool;
   //          bit13 : Bool;
   //          bit14 : Bool;
   //          bit15 : Bool;
   //          StoppedMotion : Bool;
   //          EnableDriveErr : Bool;
   //          FollowingDistErr : Bool;
   //          StandstillErr : Bool;
   //          TargetApproachErr : Bool;
   //          EncoderErr : Bool;
   //          OutputErr : Bool;
   //          ConfigErr : Bool;
   //          DriveErr : Bool;
   //          bit25 : Bool;
   //          bit26 : Bool;
   //          bit27 : Bool;
   //          bit28 : Bool;
   //          bit29 : Bool;
   //          bit30 : Bool;
   //          bit31 : Bool;
   //       END_STRUCT;
   //       Config : Struct
   //          Err_AxisLimit : Bool;
   //          Err_MaxVelocity : Bool;
   //          Err_MaxAcceleration : Bool;
   //          Err_MaxDeceleration : Bool;
   //          Err_MonTimeTargetAppr : Bool;
   //          Err_TargetRange : Bool;
   //          Err_StandstillRange : Bool;
   //          Err_MaxFollowingDist : Bool;
   //          Err_EmergencyDec : Bool;
   //          Err_StepsPerRev : Bool;
   //          Err_DisplacementPerRev : Bool;
   //          Err_NumberRevs : Bool;
   //          Err_PolarityEncoder : Bool;
   //          Err_PolarityDrive : Bool;
   //          Err_DriveInputAtMaxVel : Bool;
   //          Err_AxisLength : Bool;
   //          Err_EncoderRange : Bool;
   //          Err_MaxVelRotaryAxis : Bool;
   //          Err_DriveInputAt100 : Bool;
   //       END_STRUCT;
   //       EncoderValue : DInt;
   //       RefPoint : Real;
   //       OutVelocity : Real;
   //       LastNomPosition : Real;
   //       LastNomVelocity : Real;
   //       LastNomDeceleration : Real;
   //       InternalNomPosition : Real;
   //       InternalActPos : Real;
   //       InternalPosOffset : Real;
   //       aufl : Real;
   //       AchsLaenge : Real;
   //       AchsLaenge_DI : DInt;
   //       AbsGeberLaenge_DI : DInt;
   //       LageIstwert_DI : DInt;
   //       Coord : DInt;
   //       DoneRef : Bool;
   //       EinInitLaeuft : Bool;
   //       AusInitLaeuft : Bool;
   //       EinQuittungLaeuft : Bool;
   //       AusQuittungLaeuft : Bool;
   //       EintreiberFahrbereit : Bool;
   //       ExecRef : Int;
   //       VLastNomPosition : Real;
   //       VLastNomVelocity : Real;
   //       LastInternalPosOffset : Real;
   //       RundKorrektur : Real;
   //       LastRundKorrektur : Real;
   //       LengthUnit : String[4];
   //       InputModuleType : String[24];
   //       OutputModuleType : String[24];
   //       Init : Struct
   //          I0 : Bool;
   //          I1 : Bool;
   //          I2 : Bool;
   //          I3 : Bool;
   //          I4 : Bool;
   //          I5 : Bool;
   //          I6 : Bool;
   //          I7 : Bool;
   //          I8 : Bool;
   //          I9 : Bool;
   //          I10 : Bool;
   //          I11 : Bool;
   //          I12 : Bool;
   //          I13 : Bool;
   //          I14 : Bool;
   //          I15 : Bool;
   //          I16 : Bool;
   //          I17 : Bool;
   //          I18 : Bool;
   //          I19 : Bool;
   //          I20 : Bool;
   //          I21 : Bool;
   //          I22 : Bool;
   //          I23 : Bool;
   //          I24 : Bool;
   //          I25 : Bool;
   //          I26 : Bool;
   //          I27 : Bool;
   //          I28 : Bool;
   //          I29 : Bool;
   //          I30 : Bool;
   //          I31 : Bool;
   //       END_STRUCT;
   //    END_STRUCT;
   //    Init : Bool;
   // END_VAR
   // VAR RETAIN
   //    Raster : Bool;
   //    Bitanzahl : Int;
   //    LageDiff_R : Real;
   //    Faktor : Real;
   //    AusFaktor : Real;
   //    WertBei10V : Real;
   // END_VAR
BEGIN
END_DATA_BLOCK

